# B&R Automation Studio project DuctLines (part 14)

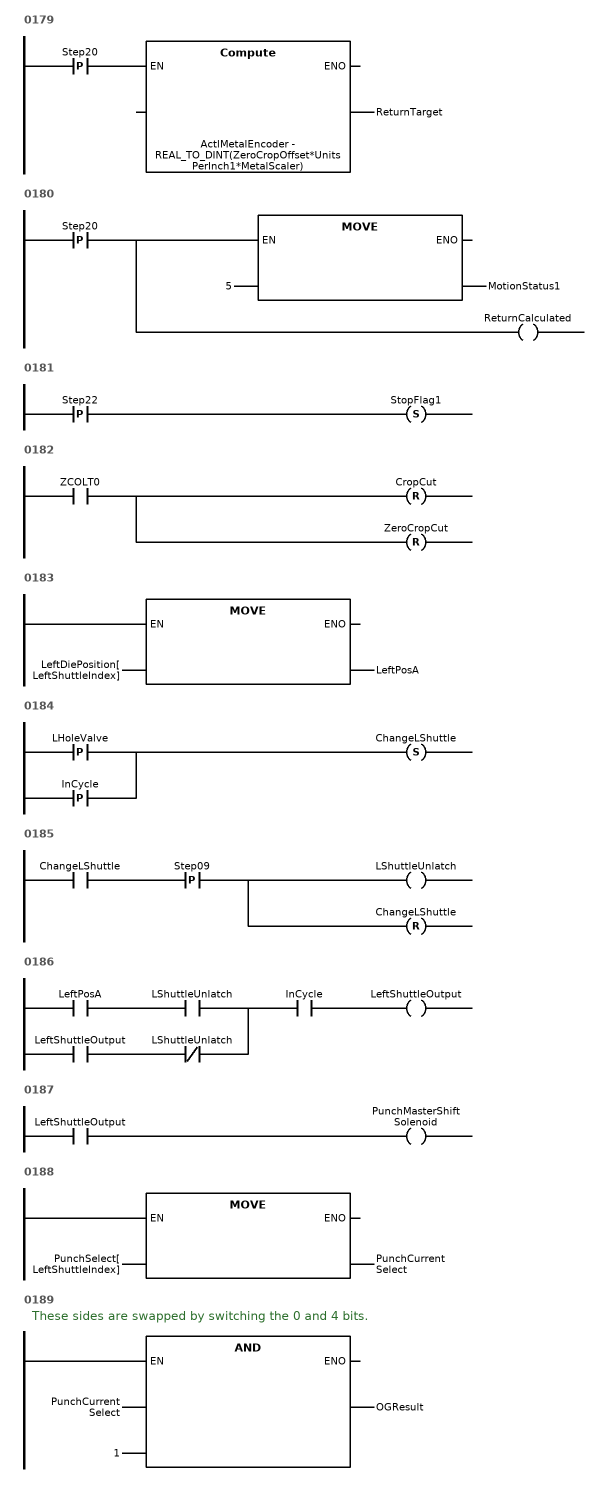
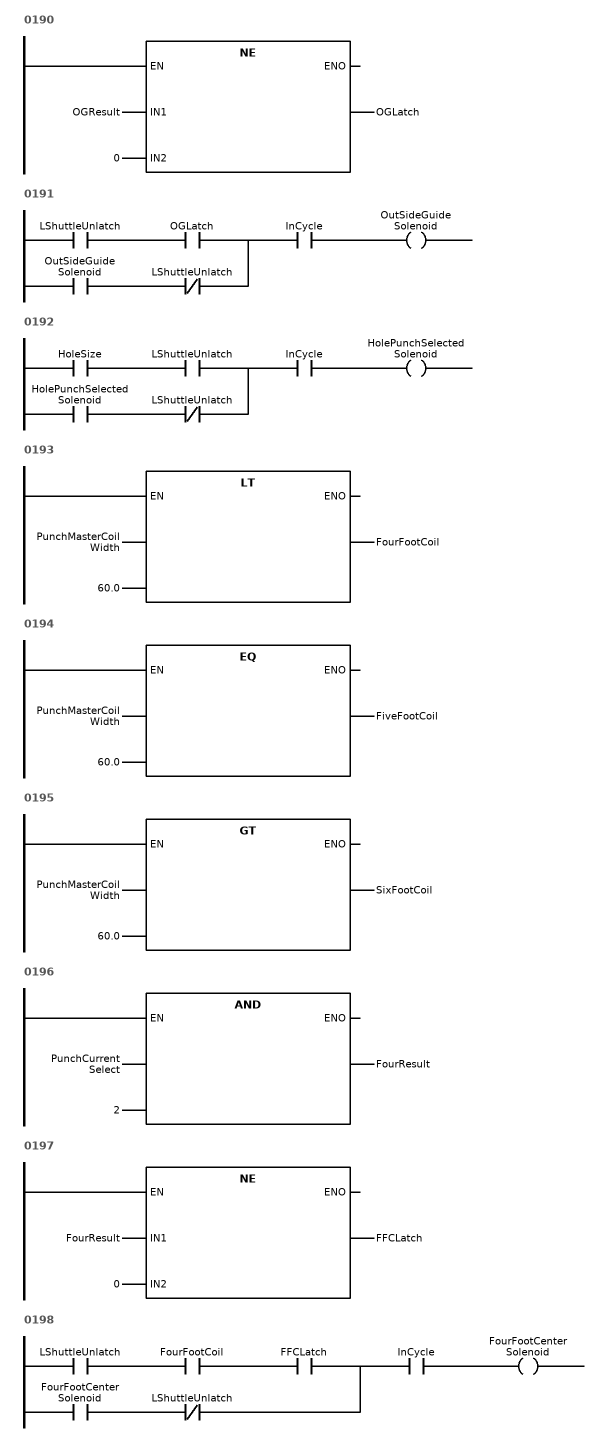
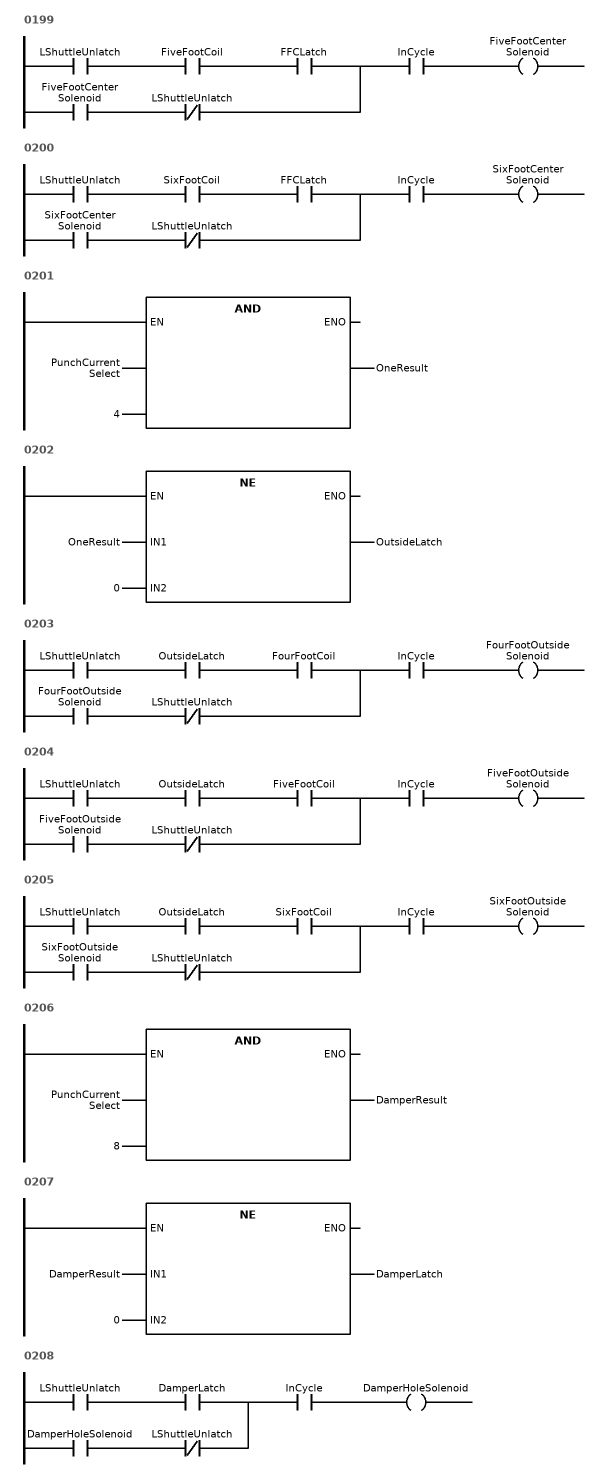
Ladder, written as Structured Text:
```iecst
PROGRAM _CYCLIC
VAR
    _e1 : R_TRIG;
    _e2 : R_TRIG;
    _e3 : R_TRIG;
    _e4 : R_TRIG;
    _e5 : F_TRIG;
    _e6 : F_TRIG;
    _e7 : R_TRIG;
    _e8 : R_TRIG;
    _e9 : R_TRIG;
    _e10 : F_TRIG;
    _e11 : F_TRIG;
    _e12 : F_TRIG;
    _e13 : R_TRIG;
    _e14 : R_TRIG;
    _e15 : F_TRIG;
    _e16 : R_TRIG;
    _e17 : R_TRIG;
    _e18 : R_TRIG;
    _e19 : R_TRIG;
    _e20 : F_TRIG;
    _e21 : F_TRIG;
    _e22 : F_TRIG;
    _e23 : R_TRIG;
    _e24 : R_TRIG;
    _e25 : R_TRIG;
    _e26 : R_TRIG;
    _e27 : R_TRIG;
    _e28 : R_TRIG;
    _e29 : R_TRIG;
    _e30 : R_TRIG;
    _e31 : R_TRIG;
    _e32 : R_TRIG;
    _e33 : R_TRIG;
    _e34 : R_TRIG;
    _e35 : F_TRIG;
    _e36 : R_TRIG;
    _e37 : R_TRIG;
    _e38 : F_TRIG;
    _e39 : R_TRIG;
    _e40 : R_TRIG;
    _e41 : R_TRIG;
    _e42 : R_TRIG;
    _e43 : F_TRIG;
    _e44 : R_TRIG;
    _e45 : F_TRIG;
    _e46 : R_TRIG;
    _e47 : F_TRIG;
    _e48 : R_TRIG;
    _e49 : F_TRIG;
    _e50 : R_TRIG;
    _e51 : F_TRIG;
    _e52 : R_TRIG;
    _e53 : F_TRIG;
    _e54 : R_TRIG;
    _e55 : F_TRIG;
    _e56 : R_TRIG;
    _e57 : F_TRIG;
    _e58 : R_TRIG;
    _e59 : F_TRIG;
    _e60 : R_TRIG;
    _e61 : F_TRIG;
    _e62 : R_TRIG;
    _e63 : F_TRIG;
    _e64 : R_TRIG;
    _e65 : R_TRIG;
    _e66 : R_TRIG;
    _e67 : R_TRIG;
    _e68 : R_TRIG;
    _e69 : F_TRIG;
    _e70 : R_TRIG;
    _e71 : R_TRIG;
    _e72 : F_TRIG;
    _e73 : R_TRIG;
    _e74 : R_TRIG;
    _p75 : BOOL;
    _e76 : R_TRIG;
    _e77 : R_TRIG;
    _e78 : R_TRIG;
    _e79 : R_TRIG;
    _p80 : BOOL;
    _e81 : F_TRIG;
    _e82 : R_TRIG;
    _e83 : R_TRIG;
    _e84 : R_TRIG;
    _e85 : R_TRIG;
    _e86 : R_TRIG;
    _e87 : R_TRIG;
    _e88 : R_TRIG;
    _e89 : R_TRIG;
END_VAR
(* Network 1 *)
MetalEncoder := ActlMetalEncoder - CoilAccumulator;

(* Network 2 *)
_e1(CLK := FSHydraulicsButton);
CLPUnlatch := _e1.Q AND CoilLinePower;

(* Network 3 *)
_e2(CLK := FSHydraulicsButton);
CoilLinePower := (_e2.Q OR CoilLinePower) AND AllSystemsOK AND NOT CLPUnlatch;

(* Network 4 *)
_e3(CLK := RollDriveEnableButton);
RollEnableUnlatch := _e3.Q AND ProcessorDriveEnable;

(* Network 5 *)
_e4(CLK := RollDriveEnableButton);
ProcessorDriveEnable := (_e4.Q OR ProcessorDriveEnable) AND NOT RollEnableUnlatch AND ProcessorDriveReady AND EStopClear;

(* Network 6 *)
ButtonStatus[20] := ProcessorDriveEnable;

(* Network 7 *)
_e5(CLK := CoilLineHalt);
_e6(CLK := InCycle);
DuctoAutoUnlatch := (_e5.Q OR (Step18B AND NOT Step19) OR (Step18 AND OneMorePart) OR ManualSignal OR _e6.Q) AND DuctoAuto;

(* Network 8 *)
_e7(CLK := CoilLineRun);
DuctoAuto := (_e7.Q OR DuctoAuto) AND NOT DuctoAutoUnlatch;

(* Network 9 *)
CoilLineRunIndicator := DuctoAuto;

(* Network 10 *)
CoilLineHaltIndicator := NOT DuctoAuto;

(* Network 11 *)
Analog1Forward := (ProcessorJogFwd AND ProcessorDriveEnable AND NOT InCycle) OR (Step04C AND NOT Step04D);

(* Network 12 *)
Analog1Reverse := (ProcessorJogRev AND ProcessorDriveEnable AND NOT InCycle) OR (Step04 AND NOT Step04B);

(* Network 13 *)
_e8(CLK := Analog1Forward);
IF _e8.Q THEN MotionStatus1 := 4; END_IF;

(* Network 14 *)
_e9(CLK := Analog1Reverse);
IF _e9.Q THEN MotionStatus1 := 5; END_IF;

(* Network 15 *)
_e10(CLK := Analog1Forward);
_e11(CLK := Analog1Reverse);
IF (_e10.Q OR _e11.Q) AND NOT StopFlag1 THEN StopFlag1 := TRUE; END_IF;

(* Network 16 *)
LevelerBrakeSolenoid := Analog1Forward OR Analog1Reverse OR ServoLoop1Closed;

(* Network 17 *)
_e12(CLK := DuctoAuto);
IF _e12.Q AND Step13 AND NOT Step14 THEN MotionStatus1 := 9; END_IF;

(* Network 18 *)
_e13(CLK := DuctoAuto);
IF _e13.Q AND Step13 AND NOT Step14 THEN MotionStatus1 := 1; END_IF;

(* Network 19: ElectricDriveEnable Output *)
ElectricDriveEnable := MotionStatus1 >= 0;

(* Network 20 *)
_e14(CLK := Step04E);
IF _e14.Q THEN MotionStatus1 := 0; END_IF;

(* Network 21 *)
ServoLoop1Closed := (MotionStatus1 >= 0) AND (MotionStatus1 <= 3);

(* Network 22 *)
_e15(CLK := InCycle);
IF _e15.Q THEN MotionStatus1 := -1; END_IF;

(* Network 23: OneMorePart logic needs To Execute Before The FeedInitiate Signal rung. *)
JobChanging := (RunJob - 1)  <> ShearJob;

(* Network 24 *)
OneMorePart := (InCycle OR (OneMorePart AND NOT FeedInitiate)) AND JobChanging AND NOT RunContinuousSignal;

(* Network 25: Feed Initiate Signal *)
_e16(CLK := CoilLineRun);
FeedInitiate := _e16.Q AND ProcessorDriveEnable AND MatlAtMeasureRoll;

(* Network 26: Verify HMI Job change request *)
IF RunJobClick AND NOT InCycle THEN NewRunJobOk := NewRunJob <= MaxRunJob; END_IF;

(* Network 27 *)
IF RunJobClick AND NewRunJobOk AND NOT InCycle THEN RunJob := NewRunJob; END_IF;

(* Network 28 *)
IF RunJobClick THEN NewRunJobOk := FALSE; END_IF;

(* Network 29 *)
IF RunJobClick THEN RunJobClick := FALSE; END_IF;

(* Network 30: Update HMI job when the shear finishes one. *)
JobsDifferent := (RunJob - 1) <> ShearJob;

(* Network 31 *)
ChangeJob1 := InCycle AND Step19 AND ShearFires AND JobsDifferent;

(* Network 32 *)
IF ChangeJob1 THEN RunJob := ShearJob + 1; END_IF;

(* Network 33 *)
_e17(CLK := FeedInitiate);
IF _e17.Q THEN NoShearHits := FALSE; END_IF;

(* Network 34: Latch BatchActive in whenever the FeedInitiate signal comes on and the Ducto Sequence isn't started. Step04 latches after PC downloads tables and resets StartSignal. Unlatch BatchActive at that point if the shear has no hits. Step19 is the last one in the Ducto sequence. If there are no shear hits, the run is finished. BatchActive unlatches and the entire sequence unlatches. *)
SHLT0 := ShearHits < 0;

(* Network 35 *)
_e18(CLK := Step04);
NoShearHits := _e18.Q AND SHLT0;

(* Network 36 *)
_e19(CLK := WarningComplete);
_e20(CLK := MatlAtMeasureRoll);
_e21(CLK := EStopClear);
_e22(CLK := ProcessorDriveEnable);
BatchCancelUnlatch := CoilLineReset OR NoShearHits OR (_e19.Q AND NOT CoilLineRun) OR _e20.Q OR _e21.Q OR _e22.Q OR Step22;

(* Network 37 *)
InCycle := ((FeedInitiate AND NOT Step01) OR InCycle) AND NOT BatchCancelUnlatch;

(* Network 38: There are 3 of these timers *)
ZRCTon(IN := Step04A AND NOT Step04B, PT := T#500ms);
ZCReverseComplete := ZRCTon.Q;

(* Network 39 *)
DDDoneTimer(IN := Step04B AND NOT Step04C, PT := T#2s);
DirectionDelayDone := DDDoneTimer.Q;

(* Network 40 *)
ZCSCTimer(IN := Step04D, PT := T#2s);
ZCSettleComplete := ZCSCTimer.Q;

(* Network 41 *)
_e23(CLK := MatlAtMeasureRoll);
IF _e23.Q AND Step04C AND NOT Step04D THEN MetalEncoderLatch := ActlMetalEncoder; END_IF;

(* Network 42 *)
_e24(CLK := Step05A);
IF _e24.Q AND NOT ZeroCropCut THEN MetalEncoderLatch := ActlMetalEncoder; END_IF;

(* Network 43: First actions in Ducto sequence, reset indexes and moves, set start signal for PC to generate die tables. *)
IF Step01 AND NOT Step02 THEN
    ShearMove := 0.0;
    LTNotchMove := 0.0;
    VNotchMove := 0.0;
    LeftHoleMove := 0.0;
    CenterHoleMove := 0.0;
    RightHoleMove := 0.0;
    PartsMade := 0;
    ShearIndex := 0;
    LTNotchIndex := 0;
    VNotchIndex := 0;
    LeftHoleIndex := 0;
    CenterHoleIndex := 0;
    RightHoleIndex := 0;
    ButtonMove := 0.0;
    ShearBrakeMove := 0.0;
    CustomLTMove := 0.0;
    CleatMove := 0.0;
    ButtonIndex := 0;
    ShearBrakeIndex := 0;
    CustomLTIndex := 0;
END_IF;

(* Network 44 *)
IF Step01 AND NOT Step02 THEN
    CleatIndex := 0;
    ButtonActual := 0;
    CustomVMove := 0.0;
    CustomVIndex := 0;
    BeadRollMove := 0.0;
    BeadRollIndex := 0;
    StartSignal := TRUE;
END_IF;

(* Network 45: The Actual Material Counter Needs To Be Initialized To ZeroCropDifference Here, too. *)
_e25(CLK := Step05A);
IF _e25.Q THEN
    ZeroCropDifference := MetalEncoderLatch - ActlMetalEncoder;
    CoilAccumulator := ZeroCropDifference;
    MetalTarget := ZeroCropDifference;
END_IF;

(* Network 46 *)
TON_1(IN := Step05A, PT := T#200ms);
PartRefOK := TON_1.Q;

(* Network 47 *)
ProcessorEncoderReset := (Step05A AND NOT Step05B) OR (ShearValve AND NOT InCycle);

(* Network 48 *)
TON_Warning(IN := Step02 AND NOT Step03, PT := WarningDelay1);
WarningComplete := TON_Warning.Q;

(* Network 49 *)
WarningHorn := Step02 AND NOT Step03;

(* Network 50: Reset variable to get ready for a new move *)
IF Step06 AND NOT Step07 THEN
    PartCutOff := FALSE;
    ShearFires := FALSE;
    IncrementalRealTarget := 0.0;
END_IF;
InitMoveSignal := Step06 AND NOT Step07;

(* Network 51: Make Sure All Data Is Updated By PC *)
HalfUpdated1 := NOT MakeShearTable AND NOT MakeLTTable AND NOT MakeVTable AND NOT MakeLHoleTable AND NOT MakeCHoleTable;

(* Network 52 *)
HalfUpdated2 := NOT MakeRHoleTable AND NOT MakeButtonTable AND NOT MakeShearBrakeTable AND NOT MakeCleatTable;

(* Network 53 *)
DataUpdated := HalfUpdated1 AND HalfUpdated2;

(* Network 54: New Connector Logic *)
_e26(CLK := Step04);
IF _e26.Q THEN SavedConnector := LatestConnector; END_IF;

(* Network 55 *)
_e27(CLK := Step08);
IF _e27.Q THEN SetConnectorChange := (LatestConnector <> SavedConnector) AND (LTNotchHits > 0); END_IF;

(* Network 56 *)
ChangeConnector := SetConnectorChange OR (ChangeConnector AND NOT LTValve AND InCycle);

(* Network 57: Net #37-40 from PicPro.  *)
MUX1:
_e28(CLK := Step08);
IF _e28.Q AND ShearUsedUp THEN
    ShearMove := MUX(K := ShearIndex, IN2 := ShearTable[0], IN3 := ShearTable[1], IN4 := ShearTable[2], IN5 := ShearTable[3], IN6 := ShearTable[4], IN7 := ShearTable[5]);
END_IF;
IF _e28.Q AND LTUsedUp THEN
    LTNotchMove := MUX(K := LTNotchIndex, IN2 := LTNotchTable[0], IN3 := LTNotchTable[1], IN4 := LTNotchTable[2], IN5 := LTNotchTable[3], IN6 := LTNotchTable[4], IN7 := LTNotchTable[5]);
END_IF;
IF _e28.Q AND VUsedUp THEN
    VNotchMove := MUX(K := VNotchIndex, IN2 := VNotchTable[0], IN3 := VNotchTable[1], IN4 := VNotchTable[2], IN5 := VNotchTable[3], IN6 := VNotchTable[4], IN7 := VNotchTable[5]);
END_IF;

(* Network 58 *)
_e29(CLK := Step08);
IF _e29.Q AND ButtonUsedUp THEN
    ButtonMove := MUX(K := ButtonIndex, IN2 := ButtonTable[0], IN3 := ButtonTable[1], IN4 := ButtonTable[2], IN5 := ButtonTable[3], IN6 := ButtonTable[4], IN7 := ButtonTable[5]);
END_IF;
IF _e29.Q AND ShearBrakeUsedUp THEN
    ShearBrakeMove := MUX(K := ShearBrakeIndex, IN2 := ShearBrakeTable[0], IN3 := ShearBrakeTable[1], IN4 := ShearBrakeTable[2], IN5 := ShearBrakeTable[3], IN6 := ShearBrakeTable[4], IN7 := ShearBrakeTable[5]);
END_IF;
IF _e29.Q AND CustomLTUsedUp THEN
    CustomLTMove := MUX(K := CustomLTIndex, IN2 := CustomLTTable[0], IN3 := CustomLTTable[1], IN4 := CustomLTTable[2], IN5 := CustomLTTable[3], IN6 := CustomLTTable[4], IN7 := CustomLTTable[5]);
END_IF;

(* Network 59 *)
_e30(CLK := Step08);
IF _e30.Q AND CleatUsedUp THEN
    CleatMove := MUX(K := CleatIndex, IN2 := CleatTable[0], IN3 := CleatTable[1], IN4 := CleatTable[2], IN5 := CleatTable[3], IN6 := CleatTable[4], IN7 := CleatTable[5]);
END_IF;
IF _e30.Q AND CustomVUsedUp THEN
    CustomVMove := MUX(K := CustomVIndex, IN2 := CustomVTable[0], IN3 := CustomVTable[1], IN4 := CustomVTable[2], IN5 := CustomVTable[3], IN6 := CustomVTable[4], IN7 := CustomVTable[5]);
END_IF;

(* Network 60: These 4 tables have too many values for the B&R mux. *)
_e31(CLK := Step08);
IF _e31.Q AND LeftHoleUsedUp THEN LeftHoleMove := LeftHoleTable[LeftHoleIndex]; END_IF;
IF _e31.Q AND CenterHoleUsedUp THEN CenterHoleMove := CenterHoleTable[CenterHoleIndex]; END_IF;
IF _e31.Q AND RightHoleUsedUp THEN RightHoleMove := RightHoleTable[RightHoleIndex]; END_IF;
IF _e31.Q AND BeadRollUsedUp THEN BeadRollMove := BeadRollTable[BeadRollIndex]; END_IF;

(* Network 61 *)
_e32(CLK := Step08);
IF _e32.Q THEN
    LeftShuttleIndex := LeftHoleIndex;
    CenterShuttleIndex := CenterHoleIndex;
    RightShuttleIndex := RightHoleIndex;
END_IF;

(* Network 62 *)
_e33(CLK := Step08);
IF _e33.Q THEN getNextMove; END_IF;

(* Network 63 *)
_e34(CLK := Step08A);
_e35(CLK := InCycle);
IF _e34.Q OR _e35.Q THEN NextMoveDone := FALSE; END_IF;

(* Network 64 *)
ShearUsedUp := ABS(ShearMove) <= InPositionBand;

(* Network 65 *)
LTUsedUp := ABS(LTNotchMove) <= InPositionBand;

(* Network 66 *)
VUsedUp := ABS(VNotchMove) <= InPositionBand;

(* Network 67 *)
LeftHoleUsedUp := ABS(LeftHoleMove) <= InPositionBand;

(* Network 68 *)
CenterHoleUsedUp := ABS(CenterHoleMove) <= InPositionBand;

(* Network 69 *)
RightHoleUsedUp := ABS(RightHoleMove) <= InPositionBand;

(* Network 70 *)
ButtonUsedUp := ABS(ButtonMove) <= InPositionBand;

(* Network 71 *)
ShearBrakeUsedUp := ABS(ShearBrakeMove) <= InPositionBand;

(* Network 72 *)
CustomLTUsedUp := ABS(CustomLTMove) <= InPositionBand;

(* Network 73 *)
CleatUsedUp := ABS(CleatMove) <= InPositionBand;

(* Network 74 *)
CustomVUsedUp := ABS(CustomVMove) <= InPositionBand;

(* Network 75 *)
BeadRollUsedUp := ABS(BeadRollMove) <= InPositionBand;

(* Network 76 *)
_e36(CLK := Step08A);
IF _e36.Q THEN UpdateTables; END_IF;

(* Network 77 *)
_e37(CLK := Step08B);
_e38(CLK := InCycle);
IF _e37.Q OR _e38.Q THEN UpdateTablesDone := FALSE; END_IF;

(* Network 78 *)
_e39(CLK := Step08B);
IF _e39.Q THEN IncrementalRealTarget := IncrementalRealTarget + SmallResult; END_IF;

(* Network 79 *)
_e40(CLK := Step08B);
NextMoveComplete := _e40.Q AND (ShearFires OR LTFires OR VFires OR LeftHoleFires OR CenterHoleFires OR RightHoleFires OR ButtonFires OR ShearBrakeFires OR CustomLTFires OR CleatFires OR CustomVFires OR BeadRollFires);

(* Network 80 *)
_e41(CLK := Step08B);
NextMoveLookAgain := _e41.Q AND NOT NextMoveComplete;

(* Network 81 *)
_e42(CLK := LTValve);
_e43(CLK := InCycle);
IF _e42.Q OR _e43.Q THEN LTFires := FALSE; END_IF;

(* Network 82 *)
_e44(CLK := VValve);
_e45(CLK := InCycle);
IF _e44.Q OR _e45.Q THEN VFires := FALSE; END_IF;

(* Network 83 *)
_e46(CLK := LHoleValve);
_e47(CLK := InCycle);
IF _e46.Q OR _e47.Q THEN LeftHoleFires := FALSE; END_IF;

(* Network 84 *)
_e48(CLK := CHoleValve);
_e49(CLK := InCycle);
IF _e48.Q OR _e49.Q THEN CenterHoleFires := FALSE; END_IF;

(* Network 85 *)
_e50(CLK := RHoleValve);
_e51(CLK := InCycle);
IF _e50.Q OR _e51.Q THEN RightHoleFires := FALSE; END_IF;

(* Network 86 *)
_e52(CLK := CycleButtons);
_e53(CLK := InCycle);
IF _e52.Q OR _e53.Q THEN ButtonFires := FALSE; END_IF;

(* Network 87 *)
_e54(CLK := CycleMaleBender);
_e55(CLK := InCycle);
IF _e54.Q OR _e55.Q THEN ShearBrakeFires := FALSE; END_IF;

(* Network 88 *)
_e56(CLK := CustomLTValve);
_e57(CLK := InCycle);
IF _e56.Q OR _e57.Q THEN CustomLTFires := FALSE; END_IF;

(* Network 89 *)
_e58(CLK := ChangeKDRolls);
_e59(CLK := InCycle);
IF _e58.Q OR _e59.Q THEN CleatFires := FALSE; END_IF;

(* Network 90 *)
_e60(CLK := CustomVValve);
_e61(CLK := InCycle);
IF _e60.Q OR _e61.Q THEN CustomVFires := FALSE; END_IF;

(* Network 91 *)
_e62(CLK := WaitCon3);
_e63(CLK := InCycle);
IF _e62.Q OR _e63.Q THEN BeadRollFires := FALSE; END_IF;

(* Network 92 *)
_e64(CLK := Step09);
IF _e64.Q THEN MetalScaler := MetalDesired / MetalActual; END_IF;
ClearEncoderSignal := _e64.Q;

(* Network 93 *)
_e65(CLK := Step10);
IF _e65.Q AND CropCut THEN RunSpeed1 := CropPercent1; END_IF;
IF _e65.Q AND NOT CropCut THEN RunSpeed1 := PercentSpeed1; END_IF;
RunSpeedCalculated := _e65.Q;

(* Network 94 *)
IF Step11 AND NOT Step12 THEN MotionStatus1 := 1; END_IF;
FeedMoveQed := Step11 AND NOT Step12;

(* Network 95 *)
WaitToFire1 := Step14 AND LTFires AND ChangeConnector;
WaitCon1 := Step14 AND FeedInitiate;

(* Network 96 *)
TON_10(IN := WaitToFire2, PT := T#50ms);
WaitCon2 := TON_10.Q;

(* Network 97 *)
_e66(CLK := InPosition1);
WaitToFire2 := (_e66.Q OR WaitToFire2) AND NOT WaitCon2;

(* Network 98 *)
WaitCon3 := Step14 AND BeadRollFires AND FeedInitiate;
WaitToFire3 := Step14 AND BeadRollFires;

(* Network 99 *)
_e67(CLK := WaitToFire3);
IF _e67.Q THEN ChangeBeadRoll := TRUE; END_IF;

(* Network 100 *)
Wait1Ready := Step14 AND ((WaitToFire1 AND WaitCon1) OR NOT WaitToFire1);
Wait2Ready := Step14 AND ((WaitToFire2 AND WaitCon2) OR NOT WaitToFire2);
Wait3Ready := Step14 AND ((WaitToFire3 AND WaitCon3) OR NOT WaitToFire3);

(* Network 101 *)
IF (Step15 AND ShearFires) OR (NOT InCycle AND CycleShear) THEN
    shearTime := DINT_TO_TIME(ShearDwell);
END_IF;

(* Network 102 *)
TP_0(IN := (Step15 AND ShearFires) OR (NOT InCycle AND CycleShear), PT := shearTime);
ShearValve := TP_0.Q;

(* Network 103 *)
IF CycleShear THEN CycleShear := FALSE; END_IF;

(* Network 104 *)
IF (Step15 AND LTFires) OR (NOT InCycle AND CycleLTDie) THEN LTTime := DINT_TO_TIME(LTDwell); END_IF;

(* Network 105 *)
TP_1(IN := (Step15 AND LTFires) OR (NOT InCycle AND CycleLTDie), PT := LTTime);
LTValve := TP_1.Q;

(* Network 106 *)
IF CycleLTDie THEN CycleLTDie := FALSE; END_IF;

(* Network 107 *)
IF (Step15 AND VFires) OR (NOT InCycle AND CycleVDie) THEN VTime := DINT_TO_TIME(VDwell); END_IF;

(* Network 108 *)
TP_2(IN := (Step15 AND VFires) OR (NOT InCycle AND CycleVDie), PT := VTime);
VValve := TP_2.Q;

(* Network 109 *)
IF CycleVDie THEN CycleVDie := FALSE; END_IF;

(* Network 110 *)
IF (Step15 AND LeftHoleFires) OR (NOT InCycle AND CycleLDie) THEN
    LeftHoleTime := DINT_TO_TIME(LHoleDwell);
END_IF;

(* Network 111 *)
TP_3(IN := (Step15 AND LeftHoleFires) OR (NOT InCycle AND CycleLDie), PT := LeftHoleTime);
LHoleValve := TP_3.Q;

(* Network 112 *)
IF CycleLDie THEN CycleLDie := FALSE; END_IF;

(* Network 113 *)
IF (Step15 AND CenterHoleFires) OR (NOT InCycle AND CycleCDie) THEN
    CenterHoleTime := DINT_TO_TIME(CHoleDwell);
END_IF;

(* Network 114 *)
TP_4(IN := (Step15 AND CenterHoleFires) OR (NOT InCycle AND CycleCDie), PT := CenterHoleTime);
CHoleValve := TP_4.Q;

(* Network 115 *)
IF (Step15 AND RightHoleFires) OR (NOT InCycle AND CycleRDie) THEN
    RightHoleTime := DINT_TO_TIME(RHoleDwell);
END_IF;

(* Network 116 *)
TP_5(IN := (Step15 AND RightHoleFires) OR (NOT InCycle AND CycleRDie), PT := RightHoleTime);
RHoleValve := TP_5.Q;

(* Network 117 *)
IF (Step15 AND CustomLTFires) OR (NOT InCycle AND CycleCustomLTDie) THEN
    CustomLTTime := DINT_TO_TIME(CustomLTDwell);
END_IF;

(* Network 118 *)
TP_6(IN := (Step15 AND CustomLTFires) OR (NOT InCycle AND CycleCustomLTDie), PT := CustomLTTime);
CustomLTValve := TP_6.Q;

(* Network 119 *)
IF (Step15 AND CustomVFires) OR (NOT InCycle AND CycleCustomVDie) THEN
    CustomVTime := DINT_TO_TIME(CustomVDwell);
END_IF;

(* Network 120 *)
TP_7(IN := (Step15 AND CustomVFires) OR (NOT InCycle AND CycleCustomVDie), PT := CustomVTime);
CustomVValve := TP_7.Q;

(* Network 121 *)
_e68(CLK := ButtonBack7);
_e69(CLK := InCycle);
UnlatchButtons := (Step15 AND _e68.Q) OR _e69.Q;

(* Network 122 *)
_e70(CLK := Step15);
CycleButtons := ((_e70.Q AND ButtonFires) OR CycleButtons) AND NOT UnlatchButtons;

(* Network 123 *)
_e71(CLK := ShearClampUpProx);
_e72(CLK := ProcessorDriveEnable);
IF ((Step15 OR ShearBrakeLatch) AND _e71.Q) OR _e72.Q THEN BrakeLatch := FALSE; END_IF;
UnlatchBender := ((Step15 OR ShearBrakeLatch) AND _e71.Q) OR _e72.Q;

(* Network 124 *)
_e73(CLK := Step15);
CycleMaleBender := ((_e73.Q AND ShearBrakeFires) OR ShearBrakeLatch OR CycleMaleBender) AND NOT UnlatchBender;

(* Network 125 *)
_e74(CLK := Step15);
ChangeKDRolls := _e74.Q AND CleatFires;

(* Network 126 *)
LeftKnockDownRoll := (ChangeKDRolls AND LeftCleatEnable AND NOT LeftKnockDownRoll) OR (LeftKnockDownRoll AND InCycle AND NOT ChangeKDRolls);

(* Network 127 *)
RightKnockDownRoll := (ChangeKDRolls AND RightCleatEnable AND NOT RightKnockDownRoll) OR (RightKnockDownRoll AND InCycle AND NOT ChangeKDRolls);

(* Network 128 *)
_p75 := NOT ShearValve AND NOT LTValve AND NOT VValve AND NOT LHoleValve;
ThirdOff1 := _p75 AND (HolePunchUp OR NOT PunchMaster);

(* Network 129 *)
ThirdOff2 := NOT CHoleValve AND NOT RHoleValve AND NOT ChangeKDRolls AND NOT CycleMaleBender;

(* Network 130 *)
ThirdOff3 := NOT CycleButtons AND NOT CustomLTValve AND NOT CustomVValve AND NOT WaitCon3;

(* Network 131 *)
_e76(CLK := Step17);
IF _e76.Q THEN DieUpTime := DINT_TO_TIME(DieUpDelay); END_IF;

(* Network 132 *)
TON_0(IN := Step17 AND NOT Step18, PT := DieUpTime);
DieDelayDone := TON_0.Q;

(* Network 133 *)
IncPartsMade := PartCutOff;

(* Network 134 *)
_e77(CLK := Step18);
IF _e77.Q THEN GTime := DINT_TO_TIME(GapTime); END_IF;

(* Network 135 *)
TP_8(IN := Step18 AND PartCutOff AND DuctoAuto, PT := GTime);
GapTP := TP_8.Q;

(* Network 136 *)
_e78(CLK := Step18);
GapPulse := GapTP OR _e78.Q;

(* Network 137 *)
_e79(CLK := Step18);
IF _e79.Q AND IncPartsMade THEN
    PartsMade := PartsMade + 1;
    RTotalInches := PartLength + RTotalInches;
END_IF;

(* Network 138 *)
IF ChangeJob1 THEN PartsMade := 0; END_IF;

(* Network 139 *)
TotalInches := RTotalInches;

(* Network 140 *)
IF ClearLengthCountSignal THEN RTotalInches := 0; END_IF;
_p80 := ClearLengthCountSignal;
IF _p80 THEN ClearLengthCountSignal := FALSE; END_IF;

(* Network 141: Set StartSignal for touchscreen. Do the warning while waiting for data. Touchscreen resets StartSignal at the tail end of the data transfer. *)
Step01 := (FeedInitiate OR Step01) AND InCycle;

(* Network 142 *)
Step02 := (StartSignal OR Step02) AND Step01;

(* Network 143 *)
Step03 := (WarningComplete OR Step03) AND Step02;

(* Network 144 *)
Step04 := (NOT StartSignal OR Step04) AND Step03;

(* Network 145: Position material for no crop cut. Latch these rungs in if crop cutting. *)
_e81(CLK := MatlAtMeasureRoll);
Step04A := (_e81.Q OR NOT ZeroCropCut OR Step04A) AND Step04;

(* Network 146 *)
Step04B := (ZCReverseComplete OR NOT ZeroCropCut OR Step04B) AND Step04A;

(* Network 147 *)
Step04C := (DirectionDelayDone OR NOT ZeroCropCut OR Step04C) AND Step04B;

(* Network 148 *)
_e82(CLK := MatlAtMeasureRoll);
Step04D := (_e82.Q OR NOT ZeroCropCut OR Step04D) AND Step04C;

(* Network 149 *)
Step04E := (ZCSettleComplete OR Step04E) AND Step04D;

(* Network 150 *)
Step05A := (ServoLoop1Closed OR Step05A) AND Step04E;

(* Network 151 *)
Step05B := (PartRefOK OR Step05B) AND Step05A;

(* Network 152: The last step in the sequence determines if the processor should stop to wait for the FeedInitiate signal. The manual signal is set if the processor needs to stop. The manual signal ujnlatches all steps past Step05B and the waits at Step05B for for FeedInitiate. The auto signal is set if the processor can continue without a FeedInitiate signal. The auto signal unlatches all steps past Step06. *)
_e83(CLK := Step05B);
Step06 := (FeedInitiate OR _e83.Q OR Step06) AND Step05B AND NOT ManualSignal;

(* Network 153 *)
Step07 := (InitMoveSignal OR Step07) AND Step06 AND NOT AutoSignal;

(* Network 154: Step08 enables the the rungs that determine the length of the next move and what to do when it completes. This will execute multiple times in some cases before it is finished. *)
Step08 := (DataUpdated OR Step08) AND Step07 AND NOT NextMoveLookAgain;

(* Network 155 *)
Step08A := (NextMoveDone OR Step08A) AND Step08;

(* Network 156 *)
Step08B := (UpdateTablesDone OR Step08B) AND Step08A;

(* Network 157 *)
Step09 := (NextMoveComplete OR Step09) AND Step08B;

(* Network 158 *)
Step10 := (ClearEncoderSignal OR Step10) AND Step09;

(* Network 159 *)
Step11 := (RunSpeedCalculated OR Step11) AND Step10;

(* Network 160 *)
Step12 := (FeedMoveQed OR Step12) AND Step11;

(* Network 161 *)
Step13 := (NOT InPosition1 OR Step13) AND Step12;

(* Network 162 *)
Step14 := (InPosition1 OR Step14) AND Step13;

(* Network 163: Dies fire when Step15 latches. Step16 latches when when a die fires or another operation begins. Step17 latches when all operations are finished. *)
Step15 := ((Wait1Ready AND Wait2Ready AND Wait3Ready) OR Step15) AND Step14;

(* Network 164 *)
Step16 := (NOT ThirdOff1 OR NOT ThirdOff2 OR NOT ThirdOff3 OR Step16) AND Step15;

(* Network 165 *)
Step17 := ((ThirdOff1 AND ThirdOff2 AND ThirdOff3) OR Step17) AND Step16;

(* Network 166 *)
Step18 := (DieDelayDone OR Step18) AND Step17;

(* Network 167 *)
Step18A := ((GapPulse AND PartCutOff AND DuctoAuto) OR NOT PartCutOff OR NOT DuctoAuto OR Step18A) AND Step18;

(* Network 168 *)
ShearHitsLTZero := ShearHits < 0;

(* Network 169 *)
Step18B := (NOT GapPulse OR ShearHitsLTZero OR NOT DuctoAuto OR Step18B) AND Step18A;

(* Network 170 *)
Step19 := (NOT ShearFires OR (ShearFires AND ((NOT MakeShearTable AND NOT OneMorePart) OR (NOT DuctoAuto AND OneMorePart))) OR Step19) AND Step18B;

(* Network 171 *)
ManualSignal := Step19 AND NOT ShearHitsLTZero AND ShearFires AND (CropCut OR (PartCutOff AND NOT DuctoAuto));
AutoSignal := Step19 AND NOT ShearHitsLTZero AND (NOT ShearFires OR (ShearFires AND ((NOT PartCutOff AND NOT CropCut) OR (PartCutOff AND DuctoAuto))));

(* Network 172 *)
Step20 := (ShearHitsLTZero OR Step20) AND Step19;

(* Network 173 *)
Step21 := (ReturnCalculated OR Step21) AND Step20;

(* Network 174 *)
ReturnComplete := ActlMetalEncoder <= ReturnTarget;

(* Network 175 *)
Step22 := (ReturnComplete OR NOT MatlAtMeasureRoll OR Step22) AND Step21;

(* Network 176 *)
IF ManualSignal AND ShearFires AND CropCut THEN CropCut := FALSE; END_IF;

(* Network 177 *)
IF NOT InCycle AND NOT CropCut THEN CropCut := TRUE; END_IF;

(* Network 178 *)
IF AutoSignal AND ZeroCropCut THEN ZCOLT0 := ZeroCropOffset <= 0; END_IF;

(* Network 179 *)
_e84(CLK := Step20);
IF _e84.Q THEN
    ReturnTarget := ActlMetalEncoder - REAL_TO_DINT(ZeroCropOffset*UnitsPerInch1*MetalScaler);
END_IF;

(* Network 180 *)
_e85(CLK := Step20);
IF _e85.Q THEN MotionStatus1 := 5; END_IF;
ReturnCalculated := _e85.Q;

(* Network 181 *)
_e86(CLK := Step22);
IF _e86.Q THEN StopFlag1 := TRUE; END_IF;

(* Network 182 *)
IF ZCOLT0 THEN
    CropCut := FALSE;
    ZeroCropCut := FALSE;
END_IF;

(* Network 183 *)
LeftPosA := LeftDiePosition[LeftShuttleIndex];

(* Network 184 *)
_e87(CLK := LHoleValve);
_e88(CLK := InCycle);
IF _e87.Q OR _e88.Q THEN ChangeLShuttle := TRUE; END_IF;

(* Network 185 *)
_e89(CLK := Step09);
LShuttleUnlatch := ChangeLShuttle AND _e89.Q;
IF ChangeLShuttle AND _e89.Q THEN ChangeLShuttle := FALSE; END_IF;

(* Network 186 *)
LeftShuttleOutput := ((LeftPosA AND LShuttleUnlatch) OR (LeftShuttleOutput AND NOT LShuttleUnlatch)) AND InCycle;

(* Network 187 *)
PunchMasterShiftSolenoid := LeftShuttleOutput;

(* Network 188 *)
PunchCurrentSelect := PunchSelect[LeftShuttleIndex];

(* Network 189: These sides are swapped by switching the 0 and 4 bits. *)
OGResult := PunchCurrentSelect AND 1;

(* Network 190 *)
OGLatch := OGResult <> 0;

(* Network 191 *)
OutSideGuideSolenoid := ((LShuttleUnlatch AND OGLatch) OR (OutSideGuideSolenoid AND NOT LShuttleUnlatch)) AND InCycle;

(* Network 192 *)
HolePunchSelectedSolenoid := ((HoleSize AND LShuttleUnlatch) OR (HolePunchSelectedSolenoid AND NOT LShuttleUnlatch)) AND InCycle;

(* Network 193 *)
FourFootCoil := PunchMasterCoilWidth < 60.0;

(* Network 194 *)
FiveFootCoil := PunchMasterCoilWidth = 60.0;

(* Network 195 *)
SixFootCoil := PunchMasterCoilWidth > 60.0;

(* Network 196 *)
FourResult := PunchCurrentSelect AND 2;

(* Network 197 *)
FFCLatch := FourResult <> 0;

(* Network 198 *)
FourFootCenterSolenoid := ((LShuttleUnlatch AND FourFootCoil AND FFCLatch) OR (FourFootCenterSolenoid AND NOT LShuttleUnlatch)) AND InCycle;

(* Network 199 *)
FiveFootCenterSolenoid := ((LShuttleUnlatch AND FiveFootCoil AND FFCLatch) OR (FiveFootCenterSolenoid AND NOT LShuttleUnlatch)) AND InCycle;

(* Network 200 *)
SixFootCenterSolenoid := ((LShuttleUnlatch AND SixFootCoil AND FFCLatch) OR (SixFootCenterSolenoid AND NOT LShuttleUnlatch)) AND InCycle;

(* Network 201 *)
OneResult := PunchCurrentSelect AND 4;

(* Network 202 *)
OutsideLatch := OneResult <> 0;

(* Network 203 *)
FourFootOutsideSolenoid := ((LShuttleUnlatch AND OutsideLatch AND FourFootCoil) OR (FourFootOutsideSolenoid AND NOT LShuttleUnlatch)) AND InCycle;

(* Network 204 *)
FiveFootOutsideSolenoid := ((LShuttleUnlatch AND OutsideLatch AND FiveFootCoil) OR (FiveFootOutsideSolenoid AND NOT LShuttleUnlatch)) AND InCycle;

(* Network 205 *)
SixFootOutsideSolenoid := ((LShuttleUnlatch AND OutsideLatch AND SixFootCoil) OR (SixFootOutsideSolenoid AND NOT LShuttleUnlatch)) AND InCycle;

(* Network 206 *)
DamperResult := PunchCurrentSelect AND 8;

(* Network 207 *)
DamperLatch := DamperResult <> 0;

(* Network 208 *)
DamperHoleSolenoid := ((LShuttleUnlatch AND DamperLatch) OR (DamperHoleSolenoid AND NOT LShuttleUnlatch)) AND InCycle;
END_PROGRAM
```

### Program Logical/DH800 (IEC)

#### Cyclic.ld
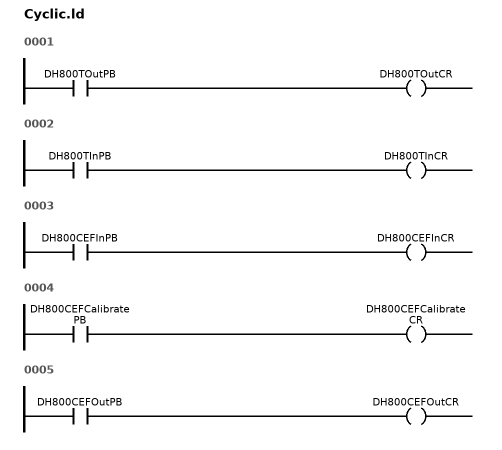
Ladder, written as Structured Text:
```iecst
PROGRAM _CYCLIC
(* Network 1 *)
DH800TOutCR := DH800TOutPB;

(* Network 2 *)
DH800TInCR := DH800TInPB;

(* Network 3 *)
DH800CEFInCR := DH800CEFInPB;

(* Network 4 *)
DH800CEFCalibrateCR := DH800CEFCalibratePB;

(* Network 5 *)
DH800CEFOutCR := DH800CEFOutPB;
END_PROGRAM
```

### Program Logical/ProgramA (IEC)

#### Variables.var
```iecst
VAR
	TON_0 : TON;
	CoilA : BOOL;
	MyEt : TIME;
END_VAR
```

#### Cyclic.ld
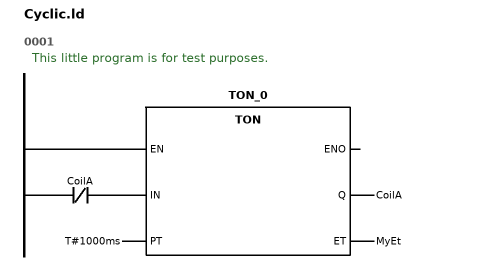
Ladder, written as Structured Text:
```iecst
PROGRAM _CYCLIC
(* Network 1: This little program is for test purposes. *)
TON_0(IN := NOT CoilA, PT := T#1000ms);
CoilA := TON_0.Q;
MyEt := TON_0.ET;
END_PROGRAM
```

### Program Logical/PMstrA (IEC)

#### Cyclic.ld
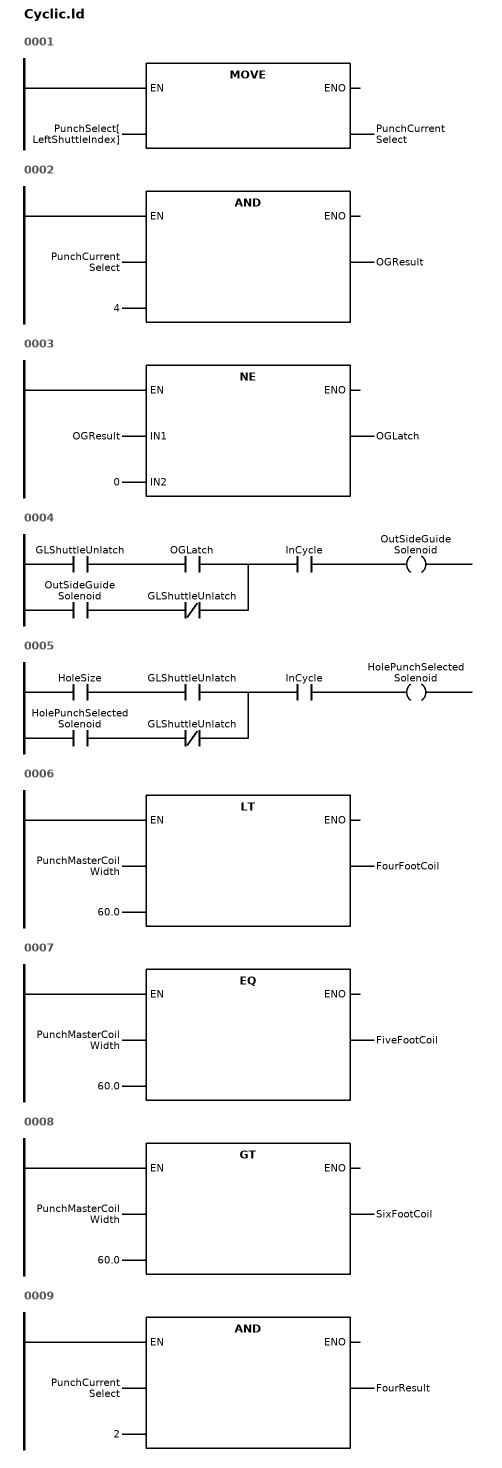
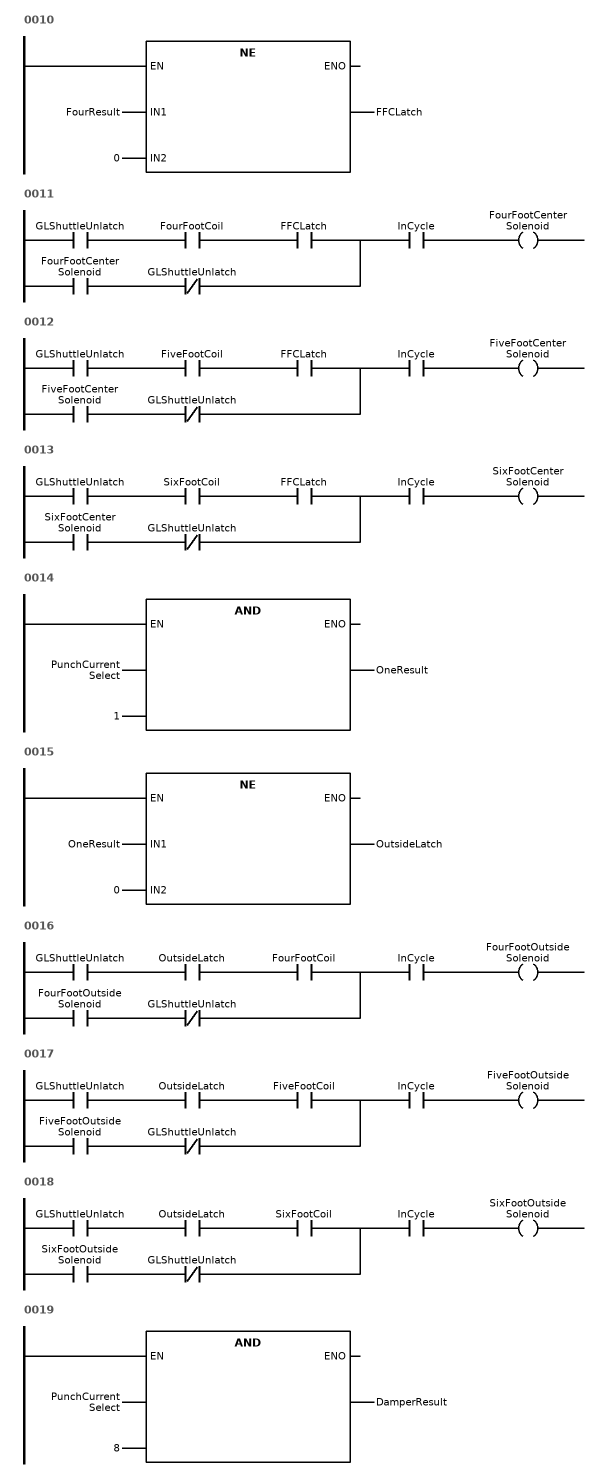
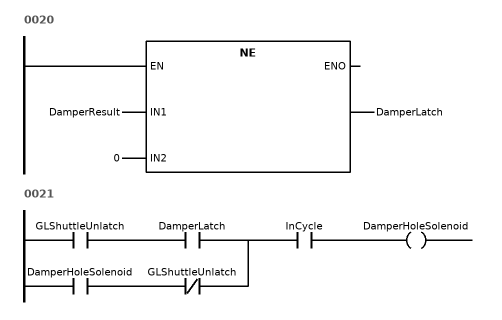
Ladder, written as Structured Text:
```iecst
PROGRAM _CYCLIC
(* Network 1 *)
PunchCurrentSelect := PunchSelect[LeftShuttleIndex];

(* Network 2 *)
OGResult := PunchCurrentSelect AND 4;

(* Network 3 *)
OGLatch := OGResult <> 0;

(* Network 4 *)
OutSideGuideSolenoid := ((GLShuttleUnlatch AND OGLatch) OR (OutSideGuideSolenoid AND NOT GLShuttleUnlatch)) AND InCycle;

(* Network 5 *)
HolePunchSelectedSolenoid := ((HoleSize AND GLShuttleUnlatch) OR (HolePunchSelectedSolenoid AND NOT GLShuttleUnlatch)) AND InCycle;

(* Network 6 *)
FourFootCoil := PunchMasterCoilWidth < 60.0;

(* Network 7 *)
FiveFootCoil := PunchMasterCoilWidth = 60.0;

(* Network 8 *)
SixFootCoil := PunchMasterCoilWidth > 60.0;

(* Network 9 *)
FourResult := PunchCurrentSelect AND 2;

(* Network 10 *)
FFCLatch := FourResult <> 0;

(* Network 11 *)
FourFootCenterSolenoid := ((GLShuttleUnlatch AND FourFootCoil AND FFCLatch) OR (FourFootCenterSolenoid AND NOT GLShuttleUnlatch)) AND InCycle;

(* Network 12 *)
FiveFootCenterSolenoid := ((GLShuttleUnlatch AND FiveFootCoil AND FFCLatch) OR (FiveFootCenterSolenoid AND NOT GLShuttleUnlatch)) AND InCycle;

(* Network 13 *)
SixFootCenterSolenoid := ((GLShuttleUnlatch AND SixFootCoil AND FFCLatch) OR (SixFootCenterSolenoid AND NOT GLShuttleUnlatch)) AND InCycle;

(* Network 14 *)
OneResult := PunchCurrentSelect AND 1;

(* Network 15 *)
OutsideLatch := OneResult <> 0;

(* Network 16 *)
FourFootOutsideSolenoid := ((GLShuttleUnlatch AND OutsideLatch AND FourFootCoil) OR (FourFootOutsideSolenoid AND NOT GLShuttleUnlatch)) AND InCycle;

(* Network 17 *)
FiveFootOutsideSolenoid := ((GLShuttleUnlatch AND OutsideLatch AND FiveFootCoil) OR (FiveFootOutsideSolenoid AND NOT GLShuttleUnlatch)) AND InCycle;

(* Network 18 *)
SixFootOutsideSolenoid := ((GLShuttleUnlatch AND OutsideLatch AND SixFootCoil) OR (SixFootOutsideSolenoid AND NOT GLShuttleUnlatch)) AND InCycle;

(* Network 19 *)
DamperResult := PunchCurrentSelect AND 8;

(* Network 20 *)
DamperLatch := DamperResult <> 0;

(* Network 21 *)
DamperHoleSolenoid := ((GLShuttleUnlatch AND DamperLatch) OR (DamperHoleSolenoid AND NOT GLShuttleUnlatch)) AND InCycle;
END_PROGRAM
```

### Program Logical/EFdrHydDrv1 (IEC) - Rungs to control an Engel processor with the original two speed hydraulic solenoids.

#### Variables.var
```iecst
VAR
	difference : DINT;
	AbsoluteDifference : DINT;
	InTargetWindow : BOOL;
	TON_0 : TON;
	MovingToPosition : BOOL;
	MoveInitiated : BOOL;
	PositionLTTarget : BOOL;
	MoveForward : BOOL;
	PositionGTTarget : BOOL;
	MoveReverse : BOOL;
	InSSWindow : BOOL;
	SettleTimerDone : BOOL;
	TP_10ms_0 : TP_10ms;
	MTPPulse : BOOL;
END_VAR
```

#### Cyclic.ld
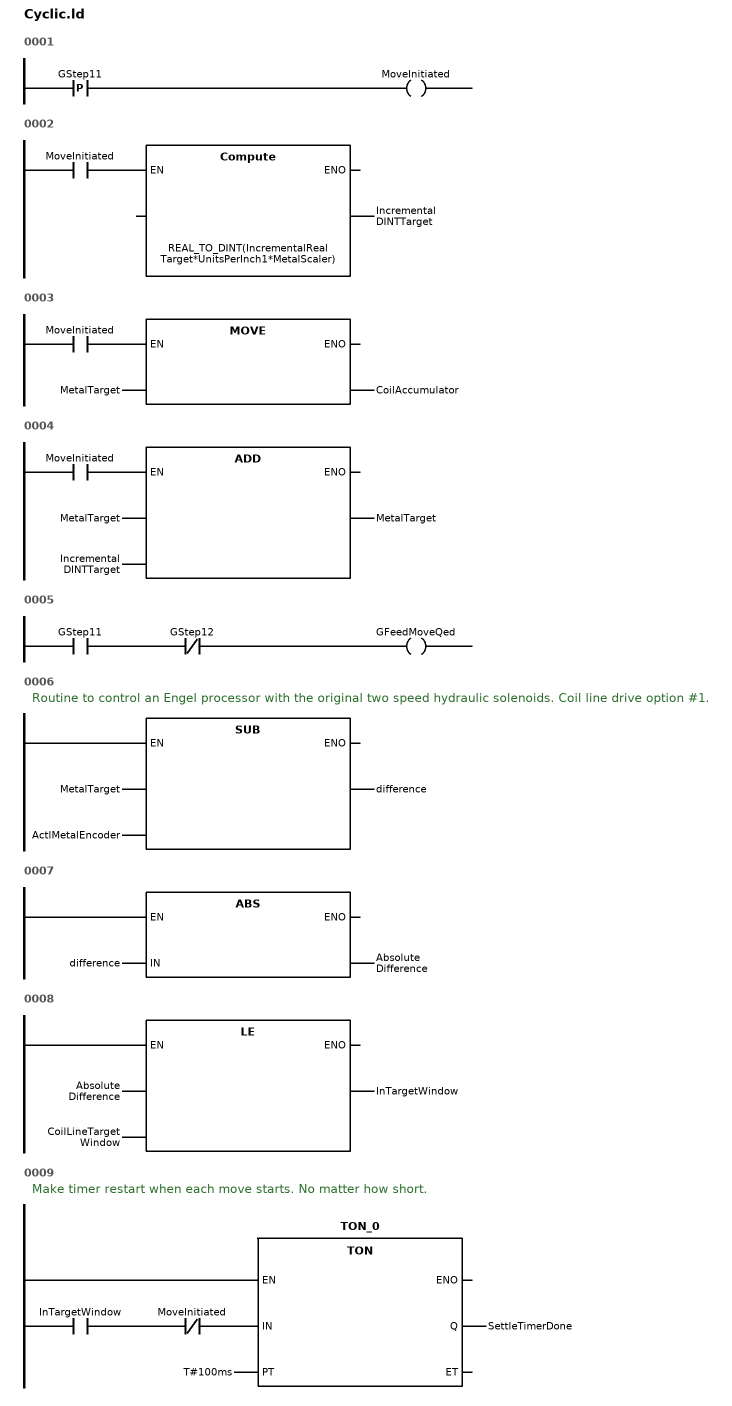
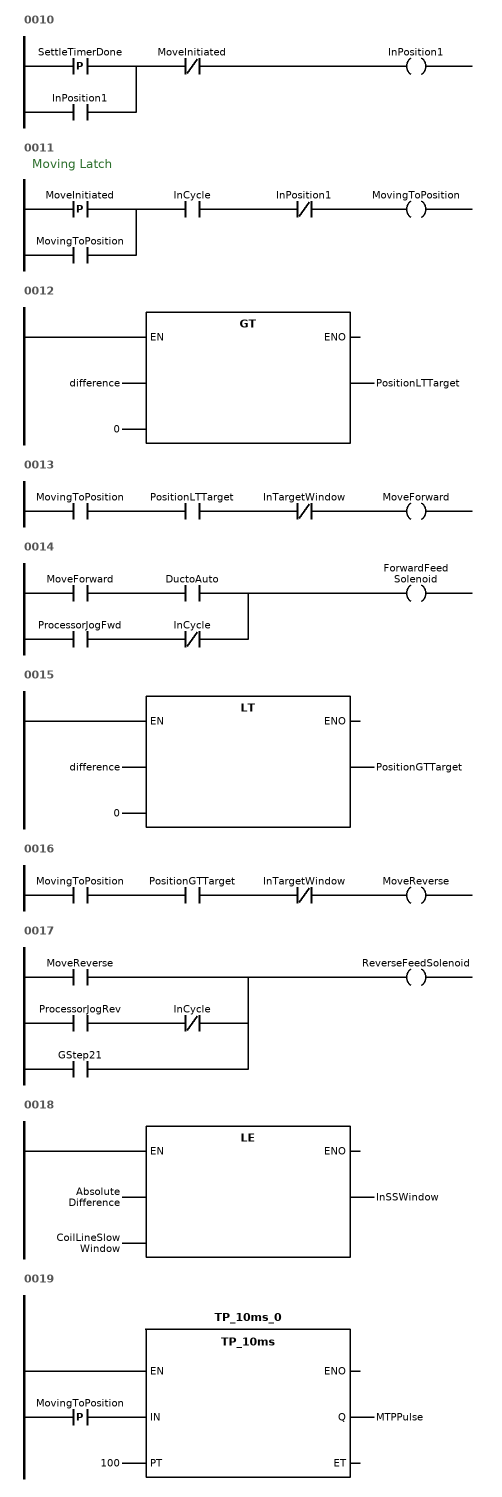
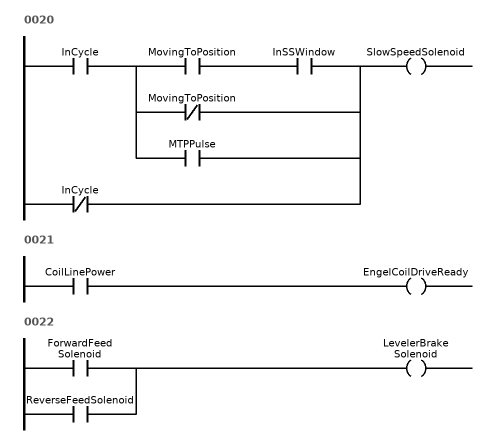
Ladder, written as Structured Text:
```iecst
PROGRAM _CYCLIC
VAR
    _e1 : R_TRIG;
    _e2 : R_TRIG;
    _e3 : R_TRIG;
    _e4 : R_TRIG;
END_VAR
(* Network 1 *)
_e1(CLK := GStep11);
MoveInitiated := _e1.Q;

(* Network 2 *)
IF MoveInitiated THEN
    IncrementalDINTTarget := REAL_TO_DINT(IncrementalRealTarget*UnitsPerInch1*MetalScaler);
END_IF;

(* Network 3 *)
IF MoveInitiated THEN CoilAccumulator := MetalTarget; END_IF;

(* Network 4 *)
IF MoveInitiated THEN MetalTarget := MetalTarget + IncrementalDINTTarget; END_IF;

(* Network 5 *)
GFeedMoveQed := GStep11 AND NOT GStep12;

(* Network 6: Routine to control an Engel processor with the original two speed hydraulic solenoids. Coil line drive option #1. *)
difference := MetalTarget - ActlMetalEncoder;

(* Network 7 *)
AbsoluteDifference := ABS(difference);

(* Network 8 *)
InTargetWindow := AbsoluteDifference <= CoilLineTargetWindow;

(* Network 9: Make timer restart when each move starts. No matter how short. *)
TON_0(IN := InTargetWindow AND NOT MoveInitiated, PT := T#100ms);
SettleTimerDone := TON_0.Q;

(* Network 10 *)
_e2(CLK := SettleTimerDone);
InPosition1 := (_e2.Q OR InPosition1) AND NOT MoveInitiated;

(* Network 11: Moving Latch *)
_e3(CLK := MoveInitiated);
MovingToPosition := (_e3.Q OR MovingToPosition) AND InCycle AND NOT InPosition1;

(* Network 12 *)
PositionLTTarget := difference > 0;

(* Network 13 *)
MoveForward := MovingToPosition AND PositionLTTarget AND NOT InTargetWindow;

(* Network 14 *)
ForwardFeedSolenoid := (MoveForward AND DuctoAuto) OR (ProcessorJogFwd AND NOT InCycle);

(* Network 15 *)
PositionGTTarget := difference < 0;

(* Network 16 *)
MoveReverse := MovingToPosition AND PositionGTTarget AND NOT InTargetWindow;

(* Network 17 *)
ReverseFeedSolenoid := MoveReverse OR (ProcessorJogRev AND NOT InCycle) OR GStep21;

(* Network 18 *)
InSSWindow := AbsoluteDifference <= CoilLineSlowWindow;

(* Network 19 *)
_e4(CLK := MovingToPosition);
TP_10ms_0(IN := _e4.Q, PT := 100);
MTPPulse := TP_10ms_0.Q;

(* Network 20 *)
SlowSpeedSolenoid := (InCycle AND ((MovingToPosition AND InSSWindow) OR NOT MovingToPosition OR MTPPulse)) OR NOT InCycle;

(* Network 21 *)
EngelCoilDriveReady := CoilLinePower;

(* Network 22 *)
LevelerBrakeSolenoid := ForwardFeedSolenoid OR ReverseFeedSolenoid;
END_PROGRAM
```

#### Init.ld
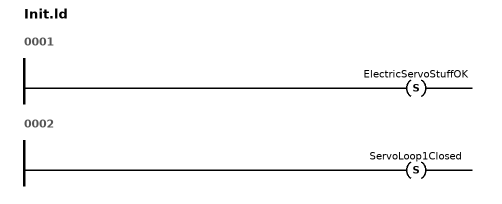
Ladder, written as Structured Text:
```iecst
PROGRAM _INIT
(* Network 1 *)
ElectricServoStuffOK := TRUE;

(* Network 2 *)
ServoLoop1Closed := TRUE;
END_PROGRAM
```

### Program Logical/Pivot_2 (IEC)

#### Variables.var
```iecst
VAR
	S1 : BOOL;
	RTCycleComplete : BOOL;
	S2 : BOOL;
	PDuctType : DINT;
	PivotPLength : REAL;
	PivotWidth : REAL;
	Residential : BOOL;
	LenLTWidth : BOOL;
	LenGTWidth : BOOL;
	TON_0 : TON;
	TON_8 : TON;
	Ton8Done : BOOL;
	S3 : BOOL;
	TON_2 : TON;
	Ton2Done : BOOL;
	S4 : BOOL;
	TON_1 : TON;
	Ton1Done : BOOL;
	S5 : BOOL;
	S6 : BOOL;
	LenGERCL : BOOL;
	PT_3 : TIME;
	TON_3 : TON;
	Ton3Done : BOOL;
	S7 : BOOL;
	S8 : BOOL;
	S9 : BOOL;
	TON_6 : TON;
	Ton6Done : BOOL;
	Jump1 : BOOL;
	S10 : BOOL;
	TON_9 : TON;
	Ton9Done : BOOL;
	S11 : BOOL;
	S12 : BOOL;
	TON_4 : TON;
	Ton4Done : BOOL;
	TON_11 : TON;
	Ton11Done : BOOL;
	S13 : BOOL;
	S14 : BOOL;
	TON_10 : TON;
	TON_5 : TON;
	Ton10Done : BOOL;
	S15 : BOOL;
END_VAR
```

#### Cyclic.ld
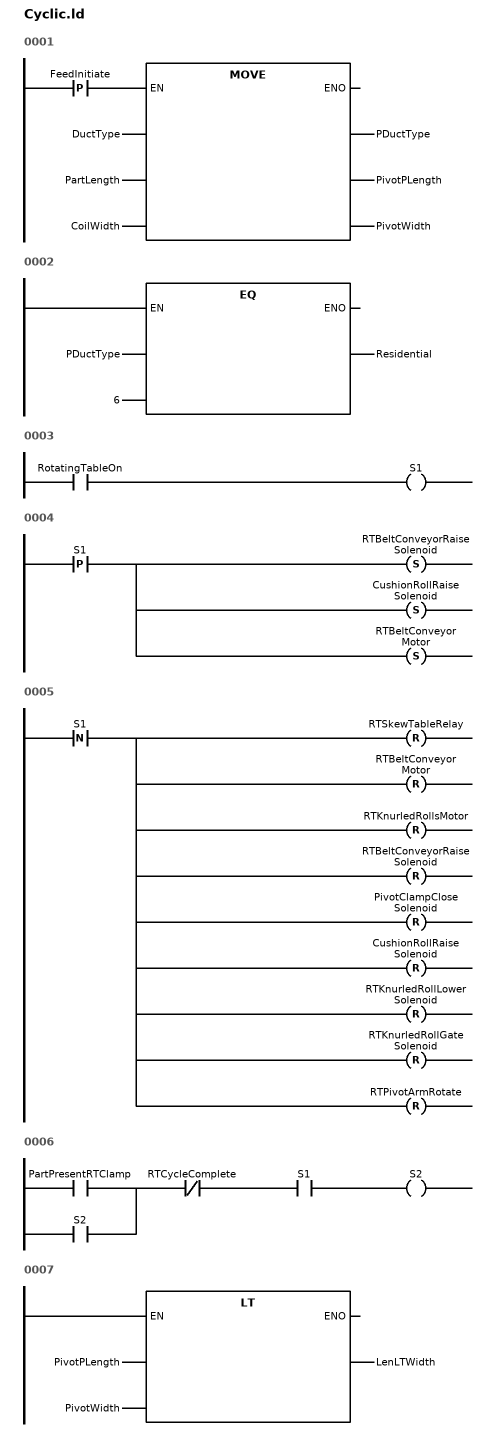
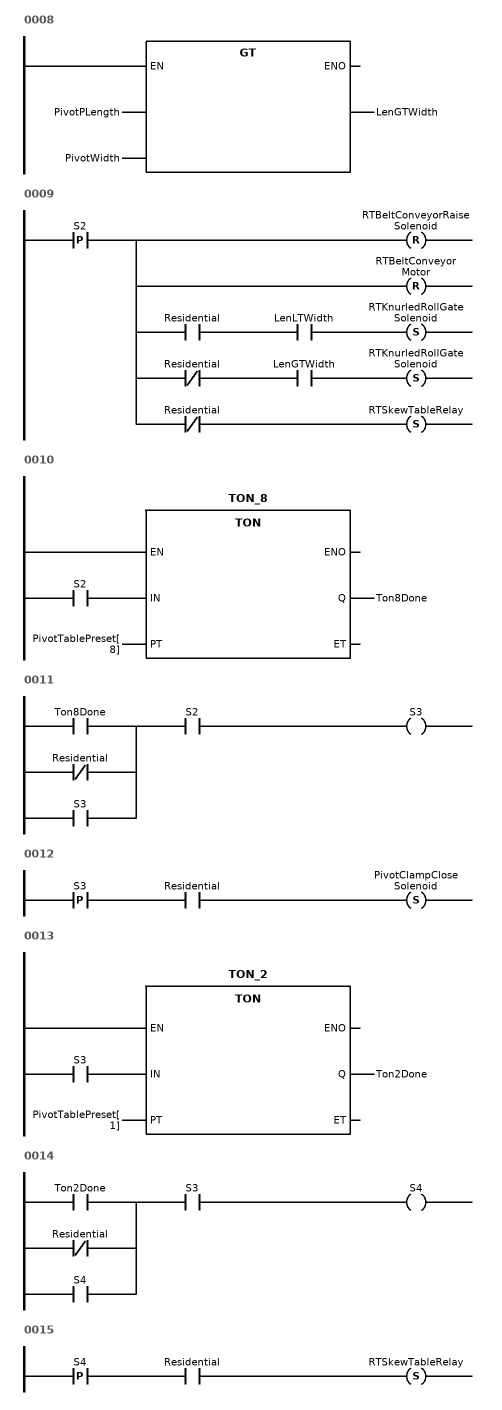
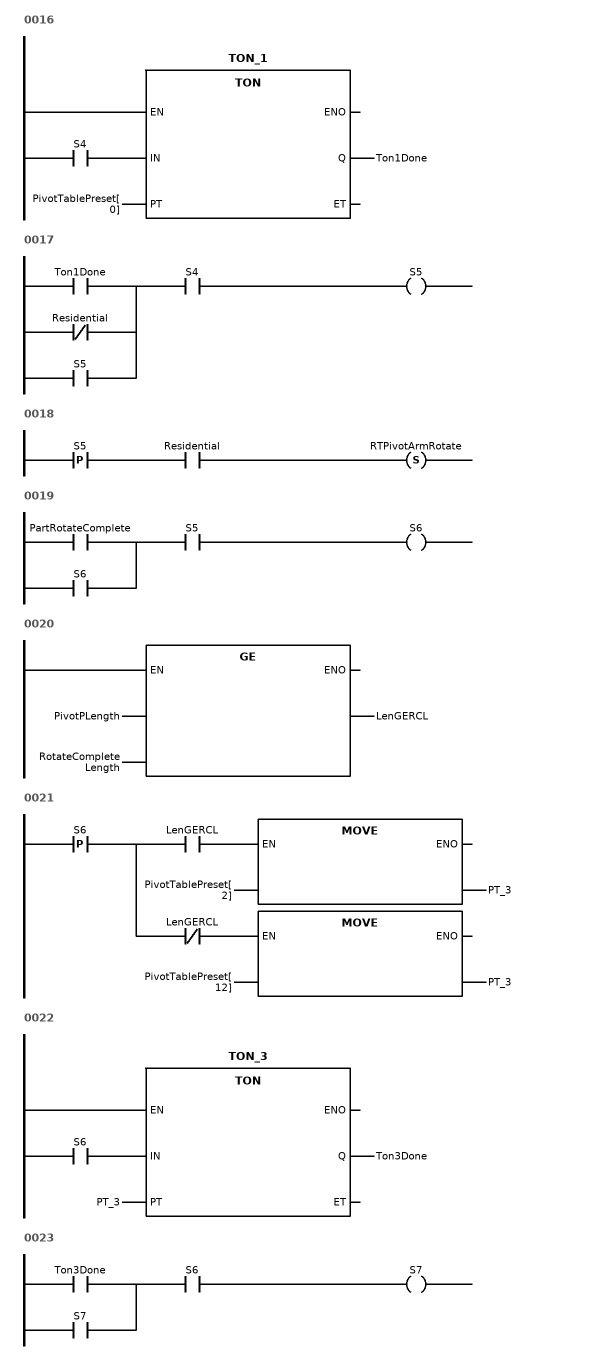
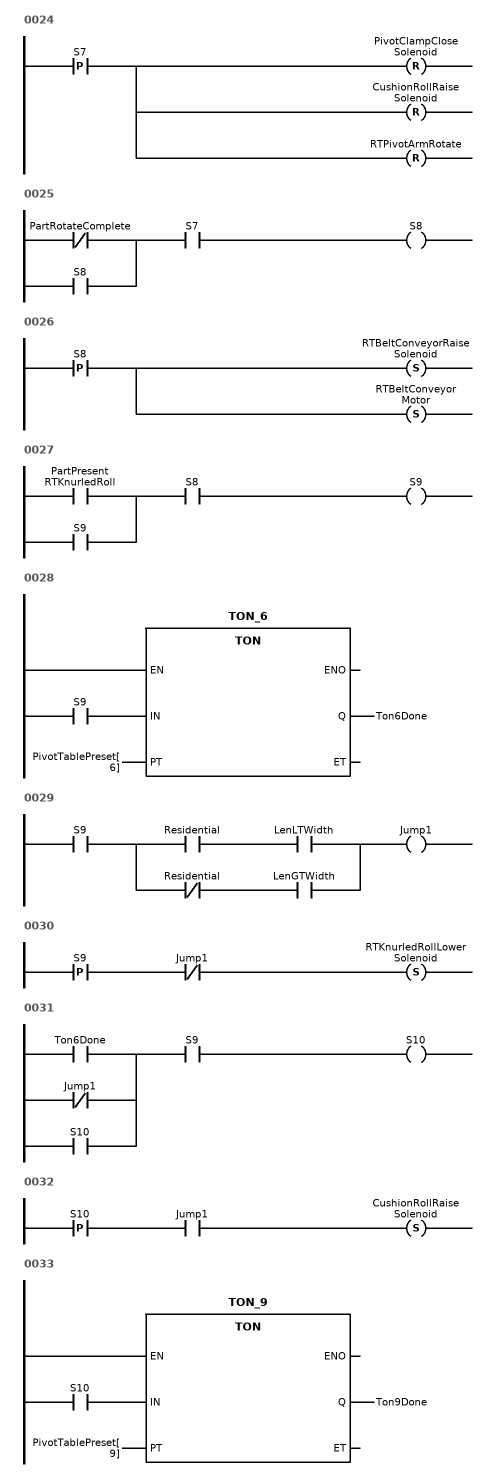
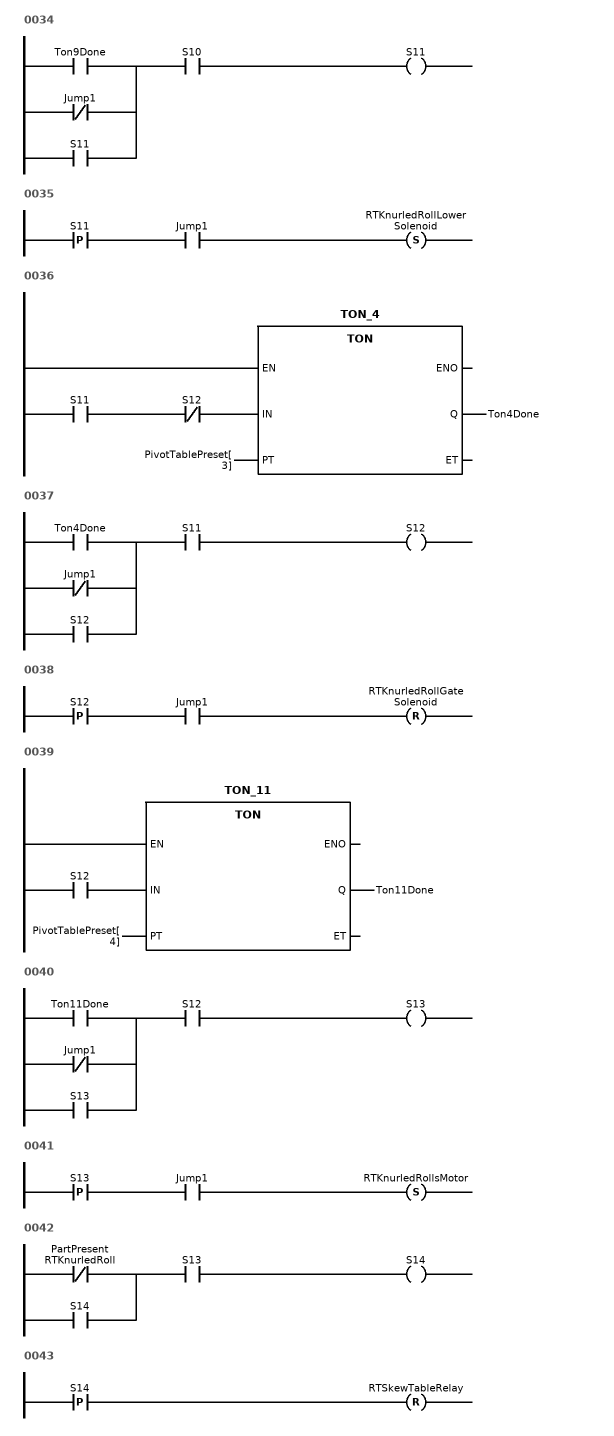
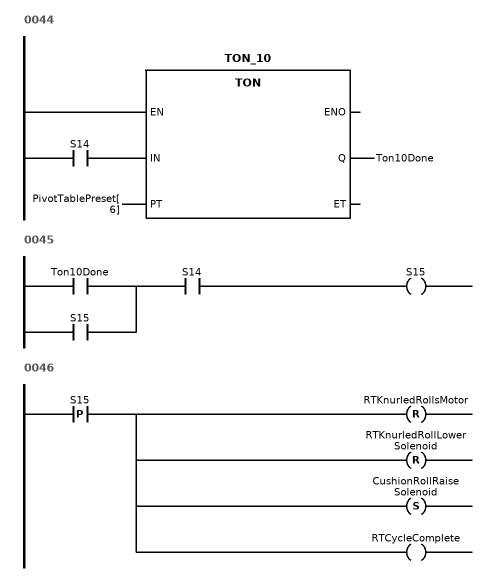
Ladder, written as Structured Text:
```iecst
PROGRAM _CYCLIC
VAR
    _e1 : R_TRIG;
    _e2 : R_TRIG;
    _e3 : F_TRIG;
    _e4 : R_TRIG;
    _e5 : R_TRIG;
    _e6 : R_TRIG;
    _e7 : R_TRIG;
    _e8 : R_TRIG;
    _e9 : R_TRIG;
    _e10 : R_TRIG;
    _e11 : R_TRIG;
    _e12 : R_TRIG;
    _e13 : R_TRIG;
    _e14 : R_TRIG;
    _e15 : R_TRIG;
    _e16 : R_TRIG;
    _e17 : R_TRIG;
END_VAR
(* Network 1 *)
_e1(CLK := FeedInitiate);
IF _e1.Q THEN
    PDuctType := DuctType;
    PivotPLength := PartLength;
    PivotWidth := CoilWidth;
END_IF;

(* Network 2 *)
Residential := PDuctType = 6;

(* Network 3 *)
S1 := RotatingTableOn;

(* Network 4 *)
_e2(CLK := S1);
IF _e2.Q THEN
    RTBeltConveyorRaiseSolenoid := TRUE;
    CushionRollRaiseSolenoid := TRUE;
    RTBeltConveyorMotor := TRUE;
END_IF;

(* Network 5 *)
_e3(CLK := S1);
IF _e3.Q THEN
    RTSkewTableRelay := FALSE;
    RTBeltConveyorMotor := FALSE;
    RTKnurledRollsMotor := FALSE;
    RTBeltConveyorRaiseSolenoid := FALSE;
    PivotClampCloseSolenoid := FALSE;
    CushionRollRaiseSolenoid := FALSE;
    RTKnurledRollLowerSolenoid := FALSE;
    RTKnurledRollGateSolenoid := FALSE;
    RTPivotArmRotate := FALSE;
END_IF;

(* Network 6 *)
S2 := (PartPresentRTClamp OR S2) AND NOT RTCycleComplete AND S1;

(* Network 7 *)
LenLTWidth := PivotPLength < PivotWidth;

(* Network 8 *)
LenGTWidth := PivotPLength > PivotWidth;

(* Network 9 *)
_e4(CLK := S2);
IF _e4.Q THEN
    RTBeltConveyorRaiseSolenoid := FALSE;
    RTBeltConveyorMotor := FALSE;
END_IF;
IF _e4.Q AND Residential AND LenLTWidth THEN RTKnurledRollGateSolenoid := TRUE; END_IF;
IF _e4.Q AND NOT Residential AND LenGTWidth THEN RTKnurledRollGateSolenoid := TRUE; END_IF;
IF _e4.Q AND NOT Residential THEN RTSkewTableRelay := TRUE; END_IF;

(* Network 10 *)
TON_8(IN := S2, PT := PivotTablePreset[8]);
Ton8Done := TON_8.Q;

(* Network 11 *)
S3 := (Ton8Done OR NOT Residential OR S3) AND S2;

(* Network 12 *)
_e5(CLK := S3);
IF _e5.Q AND Residential THEN PivotClampCloseSolenoid := TRUE; END_IF;

(* Network 13 *)
TON_2(IN := S3, PT := PivotTablePreset[1]);
Ton2Done := TON_2.Q;

(* Network 14 *)
S4 := (Ton2Done OR NOT Residential OR S4) AND S3;

(* Network 15 *)
_e6(CLK := S4);
IF _e6.Q AND Residential THEN RTSkewTableRelay := TRUE; END_IF;

(* Network 16 *)
TON_1(IN := S4, PT := PivotTablePreset[0]);
Ton1Done := TON_1.Q;

(* Network 17 *)
S5 := (Ton1Done OR NOT Residential OR S5) AND S4;

(* Network 18 *)
_e7(CLK := S5);
IF _e7.Q AND Residential THEN RTPivotArmRotate := TRUE; END_IF;

(* Network 19 *)
S6 := (PartRotateComplete OR S6) AND S5;

(* Network 20 *)
LenGERCL := PivotPLength >= RotateCompleteLength;

(* Network 21 *)
_e8(CLK := S6);
IF _e8.Q AND LenGERCL THEN PT_3 := PivotTablePreset[2]; END_IF;
IF _e8.Q AND NOT LenGERCL THEN PT_3 := PivotTablePreset[12]; END_IF;

(* Network 22 *)
TON_3(IN := S6, PT := PT_3);
Ton3Done := TON_3.Q;

(* Network 23 *)
S7 := (Ton3Done OR S7) AND S6;

(* Network 24 *)
_e9(CLK := S7);
IF _e9.Q THEN
    PivotClampCloseSolenoid := FALSE;
    CushionRollRaiseSolenoid := FALSE;
    RTPivotArmRotate := FALSE;
END_IF;

(* Network 25 *)
S8 := (NOT PartRotateComplete OR S8) AND S7;

(* Network 26 *)
_e10(CLK := S8);
IF _e10.Q THEN
    RTBeltConveyorRaiseSolenoid := TRUE;
    RTBeltConveyorMotor := TRUE;
END_IF;

(* Network 27 *)
S9 := (PartPresentRTKnurledRoll OR S9) AND S8;

(* Network 28 *)
TON_6(IN := S9, PT := PivotTablePreset[6]);
Ton6Done := TON_6.Q;

(* Network 29 *)
Jump1 := S9 AND ((Residential AND LenLTWidth) OR (NOT Residential AND LenGTWidth));

(* Network 30 *)
_e11(CLK := S9);
IF _e11.Q AND NOT Jump1 THEN RTKnurledRollLowerSolenoid := TRUE; END_IF;

(* Network 31 *)
S10 := (Ton6Done OR NOT Jump1 OR S10) AND S9;

(* Network 32 *)
_e12(CLK := S10);
IF _e12.Q AND Jump1 THEN CushionRollRaiseSolenoid := TRUE; END_IF;

(* Network 33 *)
TON_9(IN := S10, PT := PivotTablePreset[9]);
Ton9Done := TON_9.Q;

(* Network 34 *)
S11 := (Ton9Done OR NOT Jump1 OR S11) AND S10;

(* Network 35 *)
_e13(CLK := S11);
IF _e13.Q AND Jump1 THEN RTKnurledRollLowerSolenoid := TRUE; END_IF;

(* Network 36 *)
TON_4(IN := S11 AND NOT S12, PT := PivotTablePreset[3]);
Ton4Done := TON_4.Q;

(* Network 37 *)
S12 := (Ton4Done OR NOT Jump1 OR S12) AND S11;

(* Network 38 *)
_e14(CLK := S12);
IF _e14.Q AND Jump1 THEN RTKnurledRollGateSolenoid := FALSE; END_IF;

(* Network 39 *)
TON_11(IN := S12, PT := PivotTablePreset[4]);
Ton11Done := TON_11.Q;

(* Network 40 *)
S13 := (Ton11Done OR NOT Jump1 OR S13) AND S12;

(* Network 41 *)
_e15(CLK := S13);
IF _e15.Q AND Jump1 THEN RTKnurledRollsMotor := TRUE; END_IF;

(* Network 42 *)
S14 := (NOT PartPresentRTKnurledRoll OR S14) AND S13;

(* Network 43 *)
_e16(CLK := S14);
IF _e16.Q THEN RTSkewTableRelay := FALSE; END_IF;

(* Network 44 *)
TON_10(IN := S14, PT := PivotTablePreset[6]);
Ton10Done := TON_10.Q;

(* Network 45 *)
S15 := (Ton10Done OR S15) AND S14;

(* Network 46 *)
_e17(CLK := S15);
IF _e17.Q THEN
    RTKnurledRollsMotor := FALSE;
    RTKnurledRollLowerSolenoid := FALSE;
    CushionRollRaiseSolenoid := TRUE;
END_IF;
RTCycleComplete := _e17.Q;
END_PROGRAM
```

### Program Logical/CoilSelect (IEC)

#### Cyclic.ld
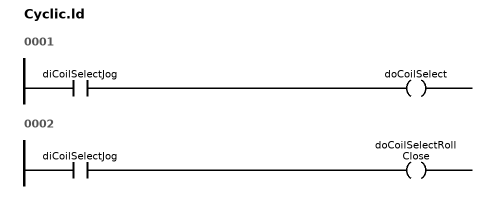
Ladder, written as Structured Text:
```iecst
PROGRAM _CYCLIC
(* Network 1 *)
doCoilSelect := diCoilSelectJog;

(* Network 2 *)
doCoilSelectRollClose := diCoilSelectJog;
END_PROGRAM
```

### Program Logical/PDButtons (IEC) - Map Soft Buttons, etc For Iowa Lines

#### Variables.var
```iecst
VAR
	PDHUnlatch : BOOL;
	hmiBrakeHydraulicsButton : BOOL;
	BHUnlatch : BOOL;
	hmiProductHydraulicsButton : BOOL;
	hmiMarkRollformerButton : BOOL;
	MROUnlatch : BOOL;
	TDCTUnlatch : BOOL;
	TDCRFMUnlatch : BOOL;
	EBeltsUnlatch : BOOL;
	hmiUncoilerOnButton : BOOL;
	UOLUnlatch : BOOL;
	hmiUncoilerLoadButton : BOOL;
	ULUnlatch : BOOL;
	hmiUncoilerRunButton : BOOL;
	URUnlatch : BOOL;
	hmiMarkTableButton : BOOL;
	MTUnlatch : BOOL;
	hmiFittingsButton : BOOL;
	hmiDuctSelectButton : BOOL;
	DSUnlatch : BOOL;
	hmiProcessorEnableButton : BOOL;
	PDEUnlatch : BOOL;
	hmiDuctoAutoButton : BOOL;
	DAUnlatch : BOOL;
	InsulmaticUnlatch : BOOL;
END_VAR
```

#### Cyclic.ld
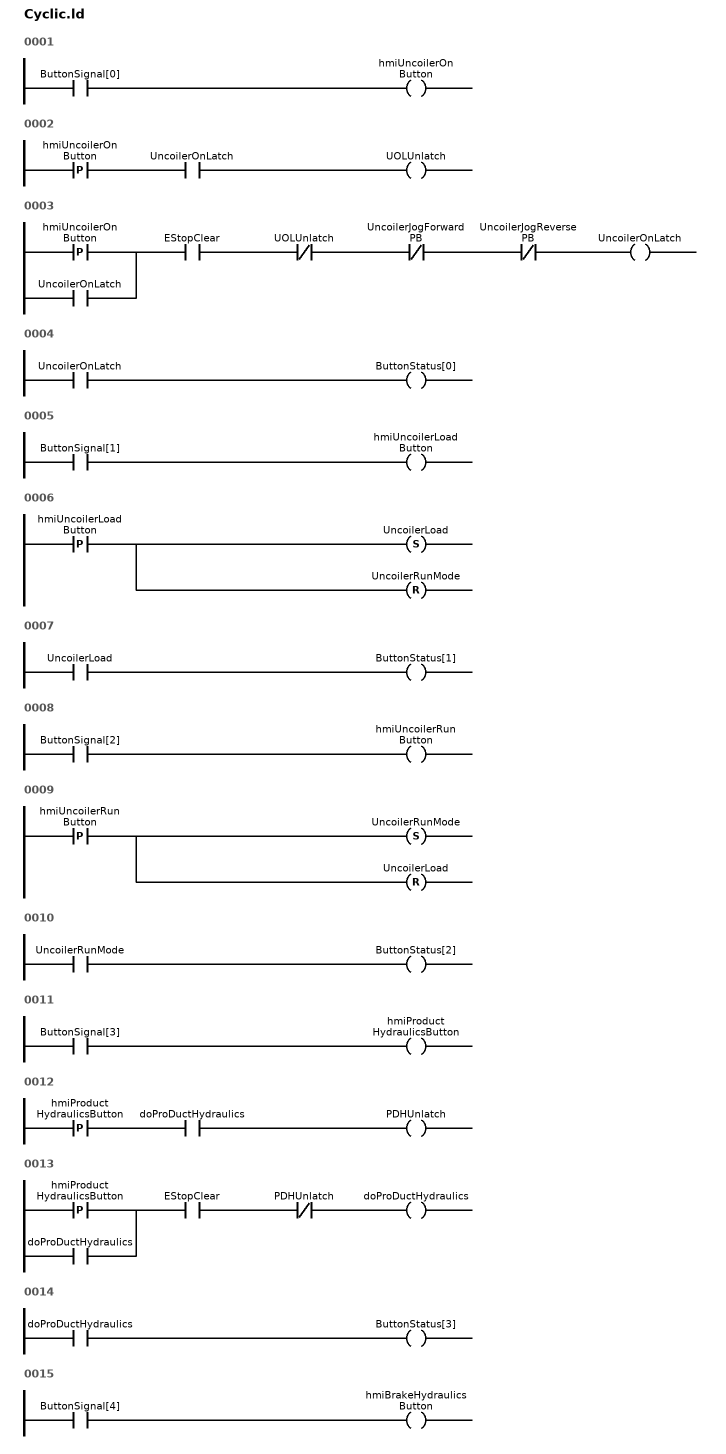
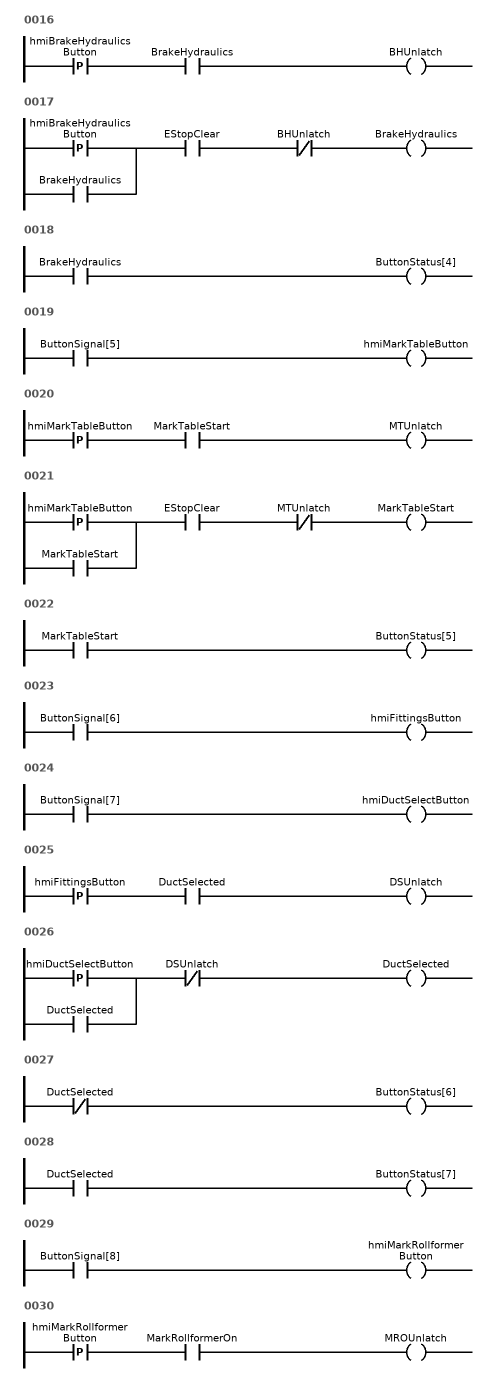
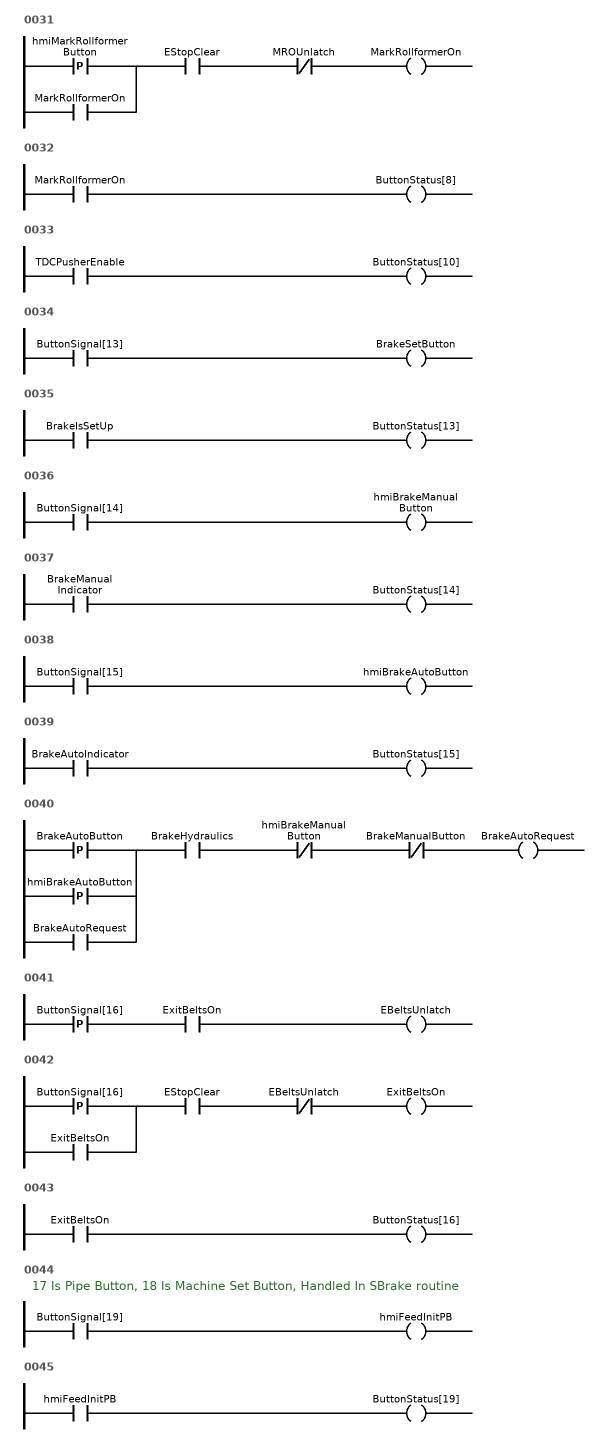
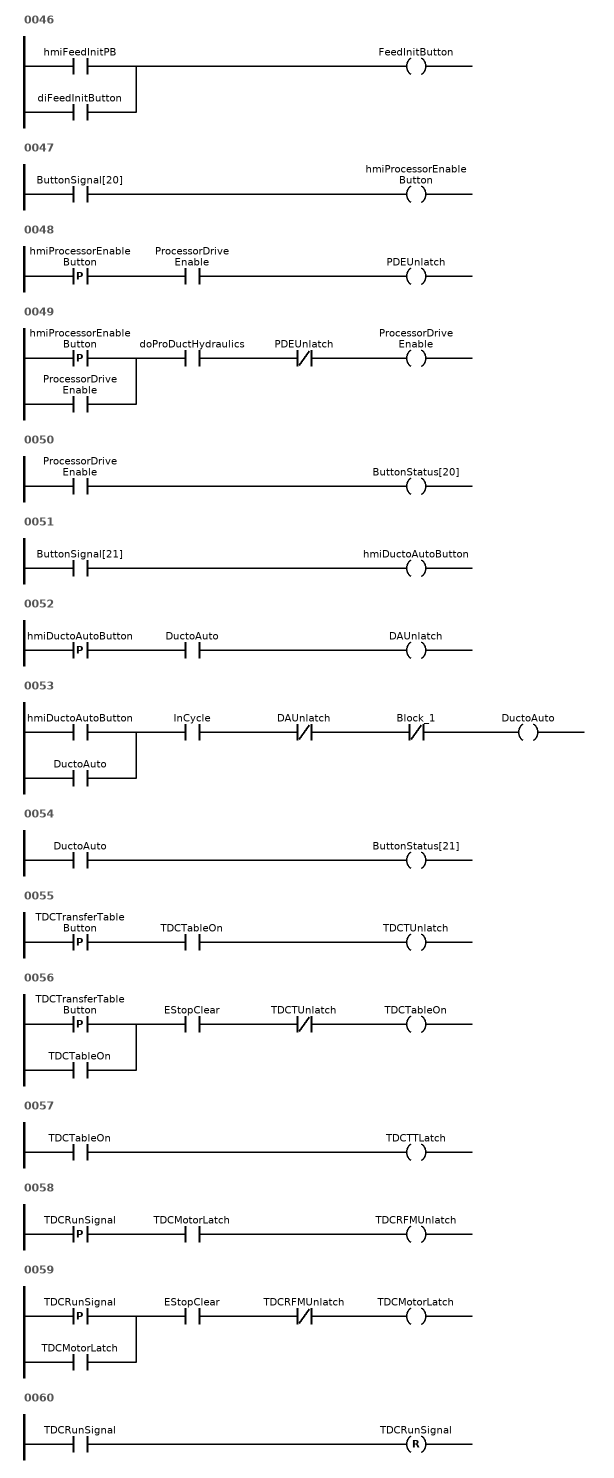
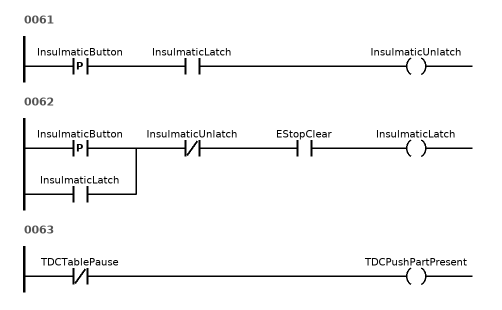
Ladder, written as Structured Text:
```iecst
PROGRAM _CYCLIC
VAR
    _e1 : R_TRIG;
    _e2 : R_TRIG;
    _e3 : R_TRIG;
    _e4 : R_TRIG;
    _e5 : R_TRIG;
    _e6 : R_TRIG;
    _e7 : R_TRIG;
    _e8 : R_TRIG;
    _e9 : R_TRIG;
    _e10 : R_TRIG;
    _e11 : R_TRIG;
    _e12 : R_TRIG;
    _e13 : R_TRIG;
    _e14 : R_TRIG;
    _e15 : R_TRIG;
    _e16 : R_TRIG;
    _e17 : R_TRIG;
    _e18 : R_TRIG;
    _e19 : R_TRIG;
    _e20 : R_TRIG;
    _e21 : R_TRIG;
    _e22 : R_TRIG;
    _e23 : R_TRIG;
    _e24 : R_TRIG;
    _e25 : R_TRIG;
    _e26 : R_TRIG;
    _e27 : R_TRIG;
END_VAR
(* Network 1 *)
hmiUncoilerOnButton := ButtonSignal[0];

(* Network 2 *)
_e1(CLK := hmiUncoilerOnButton);
UOLUnlatch := _e1.Q AND UncoilerOnLatch;

(* Network 3 *)
_e2(CLK := hmiUncoilerOnButton);
UncoilerOnLatch := (_e2.Q OR UncoilerOnLatch) AND EStopClear AND NOT UOLUnlatch AND NOT UncoilerJogForwardPB AND NOT UncoilerJogReversePB;

(* Network 4 *)
ButtonStatus[0] := UncoilerOnLatch;

(* Network 5 *)
hmiUncoilerLoadButton := ButtonSignal[1];

(* Network 6 *)
_e3(CLK := hmiUncoilerLoadButton);
IF _e3.Q THEN
    UncoilerLoad := TRUE;
    UncoilerRunMode := FALSE;
END_IF;

(* Network 7 *)
ButtonStatus[1] := UncoilerLoad;

(* Network 8 *)
hmiUncoilerRunButton := ButtonSignal[2];

(* Network 9 *)
_e4(CLK := hmiUncoilerRunButton);
IF _e4.Q THEN
    UncoilerRunMode := TRUE;
    UncoilerLoad := FALSE;
END_IF;

(* Network 10 *)
ButtonStatus[2] := UncoilerRunMode;

(* Network 11 *)
hmiProductHydraulicsButton := ButtonSignal[3];

(* Network 12 *)
_e5(CLK := hmiProductHydraulicsButton);
PDHUnlatch := _e5.Q AND doProDuctHydraulics;

(* Network 13 *)
_e6(CLK := hmiProductHydraulicsButton);
doProDuctHydraulics := (_e6.Q OR doProDuctHydraulics) AND EStopClear AND NOT PDHUnlatch;

(* Network 14 *)
ButtonStatus[3] := doProDuctHydraulics;

(* Network 15 *)
hmiBrakeHydraulicsButton := ButtonSignal[4];

(* Network 16 *)
_e7(CLK := hmiBrakeHydraulicsButton);
BHUnlatch := _e7.Q AND BrakeHydraulics;

(* Network 17 *)
_e8(CLK := hmiBrakeHydraulicsButton);
BrakeHydraulics := (_e8.Q OR BrakeHydraulics) AND EStopClear AND NOT BHUnlatch;

(* Network 18 *)
ButtonStatus[4] := BrakeHydraulics;

(* Network 19 *)
hmiMarkTableButton := ButtonSignal[5];

(* Network 20 *)
_e9(CLK := hmiMarkTableButton);
MTUnlatch := _e9.Q AND MarkTableStart;

(* Network 21 *)
_e10(CLK := hmiMarkTableButton);
MarkTableStart := (_e10.Q OR MarkTableStart) AND EStopClear AND NOT MTUnlatch;

(* Network 22 *)
ButtonStatus[5] := MarkTableStart;

(* Network 23 *)
hmiFittingsButton := ButtonSignal[6];

(* Network 24 *)
hmiDuctSelectButton := ButtonSignal[7];

(* Network 25 *)
_e11(CLK := hmiFittingsButton);
DSUnlatch := _e11.Q AND DuctSelected;

(* Network 26 *)
_e12(CLK := hmiDuctSelectButton);
DuctSelected := (_e12.Q OR DuctSelected) AND NOT DSUnlatch;

(* Network 27 *)
ButtonStatus[6] := NOT DuctSelected;

(* Network 28 *)
ButtonStatus[7] := DuctSelected;

(* Network 29 *)
hmiMarkRollformerButton := ButtonSignal[8];

(* Network 30 *)
_e13(CLK := hmiMarkRollformerButton);
MROUnlatch := _e13.Q AND MarkRollformerOn;

(* Network 31 *)
_e14(CLK := hmiMarkRollformerButton);
MarkRollformerOn := (_e14.Q OR MarkRollformerOn) AND EStopClear AND NOT MROUnlatch;

(* Network 32 *)
ButtonStatus[8] := MarkRollformerOn;

(* Network 33 *)
ButtonStatus[10] := TDCPusherEnable;

(* Network 34 *)
BrakeSetButton := ButtonSignal[13];

(* Network 35 *)
ButtonStatus[13] := BrakeIsSetUp;

(* Network 36 *)
hmiBrakeManualButton := ButtonSignal[14];

(* Network 37 *)
ButtonStatus[14] := BrakeManualIndicator;

(* Network 38 *)
hmiBrakeAutoButton := ButtonSignal[15];

(* Network 39 *)
ButtonStatus[15] := BrakeAutoIndicator;

(* Network 40 *)
_e15(CLK := BrakeAutoButton);
_e16(CLK := hmiBrakeAutoButton);
BrakeAutoRequest := (_e15.Q OR _e16.Q OR BrakeAutoRequest) AND BrakeHydraulics AND NOT hmiBrakeManualButton AND NOT BrakeManualButton;

(* Network 41 *)
_e17(CLK := ButtonSignal[16]);
EBeltsUnlatch := _e17.Q AND ExitBeltsOn;

(* Network 42 *)
_e18(CLK := ButtonSignal[16]);
ExitBeltsOn := (_e18.Q OR ExitBeltsOn) AND EStopClear AND NOT EBeltsUnlatch;

(* Network 43 *)
ButtonStatus[16] := ExitBeltsOn;

(* Network 44: 17 Is Pipe Button, 18 Is Machine Set Button, Handled In SBrake routine *)
hmiFeedInitPB := ButtonSignal[19];

(* Network 45 *)
ButtonStatus[19] := hmiFeedInitPB;

(* Network 46 *)
FeedInitButton := hmiFeedInitPB OR diFeedInitButton;

(* Network 47 *)
hmiProcessorEnableButton := ButtonSignal[20];

(* Network 48 *)
_e19(CLK := hmiProcessorEnableButton);
PDEUnlatch := _e19.Q AND ProcessorDriveEnable;

(* Network 49 *)
_e20(CLK := hmiProcessorEnableButton);
ProcessorDriveEnable := (_e20.Q OR ProcessorDriveEnable) AND doProDuctHydraulics AND NOT PDEUnlatch;

(* Network 50 *)
ButtonStatus[20] := ProcessorDriveEnable;

(* Network 51 *)
hmiDuctoAutoButton := ButtonSignal[21];

(* Network 52 *)
_e21(CLK := hmiDuctoAutoButton);
DAUnlatch := _e21.Q AND DuctoAuto;

(* Network 53 *)
DuctoAuto := (hmiDuctoAutoButton OR DuctoAuto) AND InCycle AND NOT DAUnlatch AND NOT Block_1;

(* Network 54 *)
ButtonStatus[21] := DuctoAuto;

(* Network 55 *)
_e22(CLK := TDCTransferTableButton);
TDCTUnlatch := _e22.Q AND TDCTableOn;

(* Network 56 *)
_e23(CLK := TDCTransferTableButton);
TDCTableOn := (_e23.Q OR TDCTableOn) AND EStopClear AND NOT TDCTUnlatch;

(* Network 57 *)
TDCTTLatch := TDCTableOn;

(* Network 58 *)
_e24(CLK := TDCRunSignal);
TDCRFMUnlatch := _e24.Q AND TDCMotorLatch;

(* Network 59 *)
_e25(CLK := TDCRunSignal);
TDCMotorLatch := (_e25.Q OR TDCMotorLatch) AND EStopClear AND NOT TDCRFMUnlatch;

(* Network 60 *)
IF TDCRunSignal THEN TDCRunSignal := FALSE; END_IF;

(* Network 61 *)
_e26(CLK := InsulmaticButton);
InsulmaticUnlatch := _e26.Q AND InsulmaticLatch;

(* Network 62 *)
_e27(CLK := InsulmaticButton);
InsulmaticLatch := (_e27.Q OR InsulmaticLatch) AND NOT InsulmaticUnlatch AND EStopClear;

(* Network 63 *)
TDCPushPartPresent := NOT TDCTablePause;
END_PROGRAM
```
